C07289=1093.680,277.101,420.370,177.448,19.985,152.800
C07290=1093.686,277.349,420.342,177.452,19.987,152.800
C07291=1093.691,277.598,420.313,177.455,19.990,152.800
C07292=1093.697,277.846,420.284,177.458,19.993,152.800
C07293=1093.703,278.093,420.255,177.461,19.995,152.800
C07294=1093.708,278.342,420.226,177.465,19.997,152.800
C07295=1093.714,278.591,420.197,177.468,20.000,152.800
C07296=1093.719,278.838,420.168,177.470,20.001,152.800
C07297=1093.725,279.087,420.139,177.473,20.004,152.800
C07298=1093.731,279.335,420.110,177.476,20.007,152.800
C07299=1093.737,279.584,420.081,177.480,20.009,152.800
C07300=1093.742,279.831,420.052,177.483,20.011,152.800
C07301=1093.748,280.080,420.023,177.486,20.014,152.800
C07302=1093.754,280.328,419.994,177.489,20.016,152.800
C07303=1093.759,280.576,419.965,177.493,20.018,152.800
C07304=1093.765,280.824,419.936,177.496,20.021,152.800
C07305=1093.770,281.073,419.907,177.499,20.023,152.800
C07306=1093.777,281.321,419.878,177.501,20.025,152.800
C07307=1093.781,281.569,419.849,177.505,20.028,152.800
C07308=1093.788,281.817,419.819,177.508,20.030,152.800
C07309=1093.793,282.066,419.790,177.511,20.032,152.800
C07310=1093.799,282.314,419.760,177.514,20.035,152.800
C07311=1093.804,282.561,419.732,177.517,20.038,152.800
C07312=1093.810,282.810,419.702,177.520,20.040,152.800
C07313=1093.815,283.058,419.672,177.524,20.043,152.800
C07314=1093.821,283.307,419.644,177.527,20.045,152.800
C07315=1093.826,283.555,419.615,177.530,20.047,152.800
C07316=1093.832,283.803,419.585,177.533,20.050,152.800
C07317=1093.838,284.051,419.556,177.536,20.052,152.800
C07318=1093.843,284.285,419.528,177.539,20.055,152.800
C07319=1093.849,284.520,419.501,177.542,20.057,152.800
C07320=1093.854,284.754,419.472,177.545,20.059,152.800
C07321=1093.859,284.988,419.445,177.547,20.061,152.800
C07322=1093.864,285.222,419.417,177.551,20.064,152.800
C07323=1093.870,285.456,419.389,177.554,20.066,152.800
C07324=1093.875,285.691,419.361,177.557,20.068,152.800
C07325=1093.881,285.925,419.333,177.559,20.070,152.800
C07326=1093.886,286.173,419.304,177.563,20.073,152.800
C07327=1093.892,286.421,419.274,177.566,20.076,152.800
C07328=1093.898,286.669,419.245,177.569,20.078,152.800
C07329=1093.903,286.918,419.216,177.572,20.080,152.800
C07330=1093.909,287.166,419.186,177.575,20.083,152.800
C07331=1093.915,287.414,419.156,177.578,20.085,152.800
C07332=1093.921,287.662,419.127,177.582,20.088,152.800
C07333=1093.927,287.911,419.097,177.585,20.091,152.800
C07334=1093.931,288.158,419.068,177.588,20.093,152.800
C07335=1093.937,288.407,419.038,177.591,20.095,152.800
C07336=1093.943,288.654,419.008,177.594,20.098,152.800
C07337=1093.949,288.903,418.979,177.598,20.100,152.800
C07338=1093.958,289.278,418.934,177.602,20.104,152.800
C07339=1093.966,289.653,418.888,177.607,20.108,152.801
C07340=1093.975,290.029,418.843,177.612,20.112,152.801
C07341=1093.983,290.404,418.799,177.616,20.116,152.801
C07342=1093.989,290.652,418.769,177.619,20.118,152.801
C07343=1093.994,290.900,418.739,177.623,20.121,152.801
C07344=1094.001,291.149,418.710,177.626,20.123,152.801
C07345=1094.006,291.396,418.680,177.629,20.126,152.801
C07346=1094.012,291.645,418.650,177.632,20.128,152.801
C07347=1094.018,291.893,418.620,177.635,20.131,152.801
C07348=1094.023,292.141,418.590,177.638,20.134,152.801
C07349=1094.029,292.389,418.560,177.641,20.136,152.801
C07350=1094.035,292.637,418.530,177.645,20.139,152.801
C07351=1094.040,292.885,418.500,177.648,20.141,152.801
C07352=1094.046,293.134,418.470,177.651,20.144,152.801
C07353=1094.052,293.381,418.440,177.654,20.146,152.801
C07354=1094.057,293.630,418.410,177.657,20.149,152.801
C07355=1094.063,293.878,418.380,177.660,20.152,152.801
C07356=1094.069,294.126,418.350,177.663,20.154,152.802
C07357=1094.074,294.374,418.320,177.667,20.157,152.802
C07358=1094.080,294.622,418.290,177.670,20.159,152.802
C07359=1094.086,294.870,418.260,177.673,20.162,152.802
C07360=1094.091,295.118,418.229,177.676,20.164,152.802
C07361=1094.097,295.366,418.200,177.679,20.167,152.802
C07362=1094.103,295.614,418.169,177.682,20.169,152.802
C07363=1094.109,295.862,418.139,177.685,20.172,152.802
C07364=1094.114,296.111,418.109,177.689,20.175,152.802
C07365=1094.119,296.359,418.078,177.692,20.177,152.802
C07366=1094.125,296.606,418.048,177.695,20.180,152.802
C07367=1094.131,296.855,418.018,177.698,20.183,152.802
C07368=1094.136,297.103,417.988,177.701,20.185,152.802
C07369=1094.142,297.351,417.958,177.704,20.188,152.802
C07370=1094.148,297.598,417.927,177.707,20.190,152.802
C07371=1094.154,297.846,417.897,177.710,20.193,152.802
C07372=1094.159,298.095,417.867,177.713,20.196,152.803
C07373=1094.164,298.343,417.836,177.716,20.199,152.803
C07374=1094.170,298.591,417.806,177.720,20.201,152.803
C07375=1094.176,298.838,417.776,177.723,20.204,152.803
C07376=1094.181,299.087,417.745,177.726,20.207,152.803
C07377=1094.188,299.335,417.714,177.729,20.209,152.803
C07378=1094.193,299.584,417.684,177.732,20.212,152.803
C07379=1094.198,299.832,417.653,177.735,20.215,152.803
C07380=1094.204,300.079,417.623,177.738,20.217,152.803
C07381=1094.209,300.328,417.592,177.741,20.220,152.804
C07382=1094.215,300.575,417.562,177.744,20.223,152.804
C07383=1094.221,300.823,417.531,177.748,20.226,152.804
C07384=1094.226,301.071,417.501,177.751,20.229,152.804
C07385=1094.232,301.319,417.470,177.754,20.232,152.804
C07386=1094.237,301.567,417.440,177.757,20.234,152.804
C07387=1094.242,301.815,417.409,177.760,20.237,152.804
C07388=1094.248,302.063,417.379,177.763,20.240,152.804
C07389=1094.253,302.311,417.348,177.766,20.242,152.804
C07390=1094.262,302.700,417.299,177.771,20.247,152.805
C07391=1094.271,303.089,417.251,177.776,20.251,152.805
C07392=1094.280,303.479,417.203,177.781,20.255,152.805
C07393=1094.289,303.869,417.154,177.786,20.260,152.805
C07394=1094.295,304.116,417.124,177.789,20.263,152.805
C07395=1094.300,304.365,417.093,177.792,20.266,152.805
C07396=1094.306,304.612,417.062,177.795,20.269,152.805
C07397=1094.312,304.860,417.031,177.798,20.271,152.806
C07398=1094.318,305.108,417.000,177.802,20.274,152.806
C07399=1094.323,305.357,416.969,177.804,20.277,152.806
C07400=1094.329,305.604,416.939,177.808,20.279,152.806
C07401=1094.334,305.852,416.907,177.811,20.283,152.806
C07402=1094.340,306.100,416.877,177.815,20.285,152.806
C07403=1094.346,306.349,416.846,177.817,20.288,152.806
C07404=1094.352,306.596,416.815,177.821,20.291,152.806
C07405=1094.357,306.844,416.784,177.824,20.294,152.807
C07406=1094.363,307.092,416.753,177.827,20.296,152.807
C07407=1094.369,307.340,416.721,177.830,20.299,152.807
C07408=1094.375,307.588,416.691,177.833,20.302,152.807
C07409=1094.380,307.836,416.660,177.836,20.306,152.807
C07410=1094.386,308.084,416.628,177.840,20.308,152.807
C07411=1094.391,308.332,416.598,177.843,20.311,152.807
C07412=1094.397,308.579,416.566,177.846,20.314,152.807
C07413=1094.403,308.828,416.535,177.849,20.317,152.808
C07414=1094.408,309.076,416.504,177.852,20.319,152.808
C07415=1094.414,309.323,416.473,177.855,20.322,152.808
C07416=1094.420,309.572,416.442,177.858,20.325,152.808
C07417=1094.426,309.820,416.410,177.862,20.328,152.808
C07418=1094.431,310.067,416.380,177.865,20.331,152.808
C07419=1094.437,310.316,416.348,177.868,20.334,152.808
C07420=1094.443,310.563,416.318,177.871,20.336,152.808
C07421=1094.449,310.811,416.286,177.874,20.339,152.809
C07422=1094.454,311.059,416.254,177.877,20.342,152.809
C07423=1094.460,311.307,416.224,177.880,20.345,152.809
C07424=1094.466,311.555,416.192,177.884,20.348,152.809
C07425=1094.471,311.803,416.161,177.887,20.351,152.809
C07426=1094.478,312.051,416.130,177.890,20.354,152.809
C07427=1094.483,312.299,416.097,177.893,20.357,152.809
C07428=1094.489,312.547,416.067,177.896,20.360,152.810
C07429=1094.495,312.795,416.035,177.899,20.363,152.810
C07430=1094.501,313.042,416.003,177.902,20.365,152.810
C07431=1094.506,313.291,415.972,177.906,20.369,152.810
C07432=1094.512,313.538,415.941,177.909,20.371,152.810
C07433=1094.518,313.787,415.909,177.912,20.374,152.810
C07434=1094.524,314.035,415.878,177.915,20.377,152.810
C07435=1094.530,314.283,415.847,177.918,20.380,152.811
C07436=1094.536,314.530,415.815,177.921,20.383,152.811
C07437=1094.542,314.778,415.783,177.924,20.386,152.811
C07438=1094.547,315.026,415.751,177.928,20.389,152.811
C07439=1094.553,315.274,415.721,177.931,20.392,152.811
C07440=1094.559,315.522,415.689,177.933,20.395,152.811
C07441=1094.565,315.770,415.657,177.936,20.398,152.812
C07442=1094.573,316.161,415.607,177.942,20.403,152.812
C07443=1094.582,316.554,415.556,177.947,20.408,152.812
C07444=1094.590,316.945,415.506,177.951,20.413,152.813
C07445=1094.599,317.337,415.456,177.956,20.418,152.813
C07446=1094.605,317.586,415.424,177.959,20.421,152.813
C07447=1094.611,317.833,415.392,177.962,20.424,152.813
C07448=1094.616,318.081,415.360,177.965,20.427,152.813
C07449=1094.622,318.329,415.328,177.969,20.430,152.814
C07450=1094.627,318.576,415.297,177.972,20.433,152.814
C07451=1094.633,318.825,415.265,177.975,20.436,152.814
C07452=1094.639,319.072,415.233,177.978,20.439,152.814
C07453=1094.644,319.321,415.200,177.981,20.442,152.815
C07454=1094.650,319.569,415.168,177.984,20.446,152.815
C07455=1094.655,319.816,415.137,177.987,20.449,152.815
C07456=1094.661,320.065,415.105,177.990,20.452,152.815
C07457=1094.667,320.312,415.073,177.993,20.455,152.815
C07458=1094.673,320.560,415.041,177.997,20.459,152.816
C07459=1094.678,320.808,415.009,178.000,20.462,152.816
C07460=1094.683,321.056,414.977,178.002,20.465,152.816
C07461=1094.689,321.303,414.944,178.005,20.468,152.816
C07462=1094.695,321.551,414.912,178.009,20.471,152.816
C07463=1094.701,321.800,414.880,178.012,20.474,152.817
C07464=1094.707,322.047,414.849,178.015,20.477,152.817
C07465=1094.712,322.295,414.817,178.018,20.481,152.817
C07466=1094.717,322.543,414.784,178.022,20.484,152.817
C07467=1094.723,322.791,414.752,178.024,20.487,152.818
C07468=1094.729,323.039,414.720,178.027,20.490,152.818
C07469=1094.735,323.287,414.688,178.030,20.493,152.818
C07470=1094.741,323.534,414.655,178.034,20.497,152.818
C07471=1094.746,323.783,414.623,178.037,20.500,152.819
C07472=1094.752,324.030,414.591,178.040,20.503,152.819
C07473=1094.758,324.278,414.558,178.043,20.506,152.819
C07474=1094.764,324.526,414.526,178.046,20.510,152.819
C07475=1094.769,324.774,414.494,178.049,20.513,152.820
C07476=1094.775,325.021,414.461,178.052,20.516,152.820
C07477=1094.781,325.270,414.429,178.055,20.519,152.820
C07478=1094.787,325.517,414.396,178.059,20.523,152.820
C07479=1094.792,325.765,414.364,178.062,20.526,152.820
C07480=1094.798,326.013,414.332,178.064,20.529,152.821
C07481=1094.804,326.261,414.299,178.068,20.533,152.821
C07482=1094.809,326.509,414.267,178.071,20.536,152.821
C07483=1094.815,326.756,414.234,178.074,20.539,152.821
C07484=1094.821,327.004,414.202,178.077,20.542,152.822
C07485=1094.827,327.252,414.169,178.080,20.546,152.822
C07486=1094.833,327.501,414.137,178.083,20.549,152.822
C07487=1094.838,327.747,414.105,178.086,20.552,152.822
C07488=1094.844,327.995,414.071,178.090,20.556,152.823
C07489=1094.850,328.244,414.039,178.093,20.559,152.823
C07490=1094.856,328.491,414.006,178.096,20.562,152.823
C07491=1094.861,328.740,413.974,178.099,20.566,152.823
C07492=1094.867,328.987,413.942,178.102,20.569,152.824
C07493=1094.873,329.234,413.909,178.105,20.572,152.824
C07494=1094.882,329.619,413.858,178.110,20.577,152.824
C07495=1094.891,330.004,413.807,178.115,20.583,152.825
C07496=1094.900,330.389,413.757,178.119,20.588,152.825
C07497=1094.909,330.774,413.705,178.124,20.593,152.826
C07498=1094.915,331.022,413.673,178.127,20.596,152.826
C07499=1094.921,331.269,413.640,178.131,20.600,152.826
C07500=1094.927,331.518,413.607,178.134,20.603,152.826
C07501=1094.933,331.766,413.575,178.137,20.607,152.827
C07502=1094.939,332.014,413.541,178.140,20.610,152.827
C07503=1094.945,332.261,413.508,178.143,20.614,152.827
C07504=1094.950,332.509,413.475,178.146,20.617,152.828
C07505=1094.956,332.757,413.443,178.150,20.621,152.828
C07506=1094.961,333.004,413.410,178.152,20.624,152.828
C07507=1094.967,333.252,413.377,178.156,20.628,152.829
C07508=1094.973,333.500,413.344,178.159,20.631,152.829
C07509=1094.979,333.748,413.311,178.162,20.634,152.829
C07510=1094.984,333.996,413.277,178.165,20.638,152.829
C07511=1094.991,334.243,413.245,178.168,20.642,152.830
C07512=1094.996,334.491,413.211,178.171,20.645,152.830
C07513=1095.002,334.739,413.178,178.174,20.649,152.830
C07514=1095.007,334.986,413.145,178.177,20.652,152.831
C07515=1095.013,335.234,413.112,178.181,20.656,152.831
C07516=1095.019,335.482,413.079,178.183,20.660,152.831
C07517=1095.024,335.730,413.046,178.186,20.663,152.832
C07518=1095.030,335.977,413.013,178.190,20.667,152.832
C07519=1095.036,336.225,412.980,178.192,20.670,152.832
C07520=1095.041,336.473,412.946,178.196,20.674,152.833
C07521=1095.047,336.721,412.913,178.199,20.677,152.833
C07522=1095.053,336.969,412.880,178.202,20.681,152.833
C07523=1095.059,337.216,412.846,178.205,20.685,152.834
C07524=1095.065,337.464,412.813,178.208,20.688,152.834
C07525=1095.070,337.712,412.779,178.212,20.692,152.834
C07526=1095.077,337.959,412.747,178.214,20.695,152.835
C07527=1095.082,338.207,412.713,178.217,20.699,152.835
C07528=1095.088,338.455,412.680,178.221,20.703,152.835
C07529=1095.094,338.702,412.646,178.223,20.706,152.836
C07530=1095.099,338.950,412.613,178.227,20.710,152.836
C07531=1095.105,339.198,412.579,178.230,20.714,152.836
C07532=1095.110,339.446,412.546,178.233,20.718,152.837
C07533=1095.116,339.693,412.512,178.236,20.721,152.837
C07534=1095.122,339.941,412.479,178.239,20.725,152.838
C07535=1095.128,340.189,412.446,178.242,20.729,152.838
C07536=1095.134,340.436,412.412,178.245,20.732,152.838
C07537=1095.139,340.684,412.378,178.248,20.736,152.839
C07538=1095.145,340.932,412.345,178.251,20.740,152.839
C07539=1095.151,341.179,412.311,178.254,20.744,152.840
C07540=1095.156,341.427,412.278,178.257,20.747,152.840
C07541=1095.162,341.674,412.244,178.261,20.751,152.840
C07542=1095.168,341.922,412.210,178.263,20.755,152.841
C07543=1095.174,342.170,412.176,178.267,20.759,152.841
C07544=1095.180,342.418,412.142,178.269,20.763,152.841
C07545=1095.186,342.666,412.108,178.273,20.767,152.842
C07546=1095.194,343.045,412.057,178.278,20.773,152.843
C07547=1095.203,343.424,412.005,178.282,20.778,152.843
C07548=1095.212,343.803,411.954,178.287,20.784,152.844
C07549=1095.220,344.181,411.902,178.291,20.790,152.844
C07550=1095.226,344.429,411.868,178.295,20.794,152.845
C07551=1095.232,344.677,411.834,178.297,20.798,152.845
C07552=1095.238,344.924,411.800,178.301,20.802,152.845
C07553=1095.244,345.172,411.766,178.304,20.806,152.846
C07554=1095.249,345.420,411.733,178.307,20.810,152.846
C07555=1095.255,345.667,411.699,178.310,20.813,152.847
C07556=1095.261,345.914,411.665,178.313,20.817,152.847
C07557=1095.267,346.163,411.630,178.316,20.821,152.848
C07558=1095.272,346.410,411.596,178.319,20.826,152.848
C07559=1095.278,346.658,411.562,178.322,20.829,152.849
C07560=1095.284,346.905,411.528,178.325,20.833,152.849
C07561=1095.290,347.152,411.494,178.328,20.837,152.849
C07562=1095.295,347.401,411.460,178.331,20.841,152.850
C07563=1095.301,347.649,411.426,178.335,20.846,152.850
C07564=1095.307,347.896,411.392,178.337,20.849,152.851
C07565=1095.313,348.143,411.358,178.341,20.853,152.851
C07566=1095.318,348.391,411.323,178.343,20.857,152.852
C07567=1095.324,348.638,411.289,178.347,20.862,152.852
C07568=1095.330,348.887,411.255,178.349,20.865,152.852
C07569=1095.335,349.134,411.221,178.353,20.869,152.853
C07570=1095.341,349.381,411.187,178.355,20.873,152.853
C07571=1095.347,349.629,411.153,178.359,20.878,152.854
C07572=1095.352,349.877,411.118,178.362,20.882,152.854
C07573=1095.358,350.124,411.084,178.365,20.886,152.855
C07574=1095.364,350.372,411.050,178.368,20.890,152.855
C07575=1095.369,350.619,411.015,178.371,20.894,152.856
C07576=1095.376,350.867,410.981,178.374,20.898,152.856
C07577=1095.382,351.114,410.946,178.378,20.902,152.857
C07578=1095.387,351.362,410.912,178.380,20.906,152.857
C07579=1095.393,351.609,410.878,178.383,20.911,152.858
C07580=1095.399,351.857,410.843,178.386,20.915,152.858
C07581=1095.404,352.104,410.808,178.389,20.919,152.859
C07582=1095.410,352.352,410.774,178.393,20.923,152.859
C07583=1095.416,352.600,410.739,178.395,20.927,152.860
C07584=1095.422,352.847,410.705,178.399,20.931,152.860
C07585=1095.428,353.094,410.671,178.401,20.935,152.861
C07586=1095.433,353.343,410.636,178.405,20.940,152.861
C07587=1095.440,353.589,410.601,178.408,20.944,152.862
C07588=1095.445,353.837,410.566,178.410,20.948,152.862
C07589=1095.451,354.085,410.532,178.414,20.953,152.863
C07590=1095.456,354.333,410.497,178.416,20.957,152.863
C07591=1095.463,354.579,410.463,178.420,20.961,152.864
C07592=1095.468,354.828,410.428,178.423,20.966,152.864
C07593=1095.473,355.075,410.393,178.425,20.970,152.865
C07594=1095.480,355.322,410.358,178.429,20.974,152.865
C07595=1095.485,355.570,410.323,178.432,20.978,152.866
C07596=1095.491,355.817,410.289,178.434,20.983,152.867
C07597=1095.497,356.064,410.254,178.438,20.987,152.867
C07598=1095.505,356.447,410.200,178.442,20.994,152.868
C07599=1095.514,356.828,410.146,178.447,21.000,152.869
C07600=1095.524,357.209,410.093,178.452,21.008,152.870
C07601=1095.532,357.590,410.039,178.457,21.014,152.870
C07602=1095.538,357.838,410.003,178.459,21.018,152.871
C07603=1095.544,358.085,409.969,178.462,21.023,152.872
C07604=1095.550,358.333,409.934,178.465,21.027,152.872
C07605=1095.555,358.580,409.899,178.468,21.031,152.873
C07606=1095.561,358.827,409.864,178.471,21.036,152.873
C07607=1095.567,359.075,409.829,178.475,21.040,152.874
C07608=1095.573,359.322,409.794,178.478,21.045,152.874
C07609=1095.579,359.570,409.759,178.480,21.050,152.875
C07610=1095.584,359.817,409.724,178.483,21.054,152.876
C07611=1095.590,360.065,409.688,178.487,21.059,152.876
C07612=1095.596,360.312,409.653,178.489,21.063,152.877
C07613=1095.602,360.560,409.619,178.492,21.067,152.877
C07614=1095.608,360.807,409.583,178.496,21.072,152.878
C07615=1095.614,361.055,409.547,178.499,21.077,152.879
C07616=1095.619,361.302,409.513,178.501,21.081,152.879
C07617=1095.625,361.550,409.477,178.504,21.086,152.880
C07618=1095.630,361.797,409.442,178.507,21.091,152.880
C07619=1095.637,362.044,409.407,178.510,21.095,152.881
C07620=1095.643,362.291,409.371,178.513,21.099,152.882
C07621=1095.648,362.539,409.336,178.516,21.104,152.882
C07622=1095.654,362.786,409.301,178.520,21.109,152.883
C07623=1095.660,363.034,409.265,178.522,21.113,152.883
C07624=1095.665,363.281,409.230,178.525,21.118,152.884
C07625=1095.672,363.528,409.195,178.528,21.123,152.885
C07626=1095.677,363.775,409.159,178.532,21.128,152.885
C07627=1095.683,364.023,409.124,178.534,21.132,152.886
C07628=1095.689,364.271,409.088,178.537,21.137,152.887
C07629=1095.695,364.518,409.052,178.540,21.142,152.887
C07630=1095.701,364.765,409.017,178.543,21.146,152.888
C07631=1095.706,365.012,408.981,178.546,21.152,152.889
C07632=1095.712,365.260,408.946,178.549,21.156,152.889
C07633=1095.718,365.507,408.910,178.552,21.161,152.890
C07634=1095.724,365.755,408.875,178.555,21.165,152.891
C07635=1095.730,366.002,408.839,178.558,21.170,152.891
C07636=1095.735,366.249,408.803,178.560,21.175,152.892
C07637=1095.741,366.497,408.768,178.564,21.180,152.893
C07638=1095.747,366.744,408.732,178.567,21.185,152.893
C07639=1095.753,366.992,408.697,178.570,21.190,152.894
C07640=1095.758,367.239,408.661,178.573,21.195,152.895
C07641=1095.764,367.486,408.626,178.575,21.199,152.895
C07642=1095.770,367.734,408.588,178.578,21.204,152.896
C07643=1095.775,367.981,408.553,178.581,21.209,152.897
C07644=1095.781,368.228,408.517,178.585,21.214,152.897
C07645=1095.787,368.476,408.482,178.588,21.219,152.898
C07646=1095.793,368.723,408.446,178.591,21.224,152.899
C07647=1095.799,368.970,408.410,178.593,21.229,152.900
C07648=1095.805,369.217,408.374,178.596,21.234,152.900
C07649=1095.810,369.465,408.338,178.599,21.239,152.901
C07650=1095.820,369.861,408.280,178.604,21.247,152.902
C07651=1095.829,370.258,408.223,178.609,21.255,152.903
C07652=1095.838,370.655,408.165,178.613,21.263,152.905
C07653=1095.848,371.051,408.107,178.618,21.271,152.906
C07654=1095.854,371.298,408.071,178.621,21.276,152.907
C07655=1095.859,371.545,408.035,178.624,21.281,152.907
C07656=1095.865,371.793,407.999,178.627,21.287,152.908
C07657=1095.871,372.040,407.963,178.630,21.291,152.909
C07658=1095.877,372.287,407.927,178.633,21.297,152.910
C07659=1095.882,372.534,407.890,178.635,21.301,152.910
C07660=1095.888,372.782,407.854,178.638,21.307,152.911
C07661=1095.895,373.029,407.818,178.641,21.312,152.912
C07662=1095.901,373.276,407.782,178.644,21.317,152.913
C07663=1095.906,373.524,407.745,178.647,21.322,152.913
C07664=1095.912,373.771,407.710,178.650,21.327,152.914
C07665=1095.918,374.018,407.673,178.653,21.333,152.915
C07666=1095.924,374.265,407.636,178.656,21.338,152.916
C07667=1095.930,374.513,407.601,178.659,21.343,152.916
C07668=1095.935,374.759,407.565,178.662,21.349,152.917
C07669=1095.941,375.006,407.528,178.665,21.354,152.918
C07670=1095.947,375.254,407.491,178.667,21.359,152.919
C07671=1095.953,375.502,407.455,178.670,21.364,152.920
C07672=1095.958,375.748,407.419,178.673,21.369,152.921
C07673=1095.964,375.995,407.382,178.676,21.375,152.922
C07674=1095.970,376.242,407.345,178.679,21.380,152.922
C07675=1095.976,376.490,407.309,178.682,21.386,152.923
C07676=1095.982,376.737,407.272,178.685,21.391,152.924
C07677=1095.987,376.984,407.236,178.688,21.397,152.925
C07678=1095.993,377.231,407.199,178.691,21.402,152.926
C07679=1095.999,377.478,407.162,178.693,21.408,152.927
C07680=1096.005,377.725,407.126,178.696,21.413,152.927
C07681=1096.011,377.973,407.089,178.699,21.418,152.928
C07682=1096.017,378.220,407.052,178.702,21.424,152.929
C07683=1096.022,378.467,407.016,178.705,21.429,152.930
C07684=1096.027,378.715,406.979,178.708,21.435,152.931
C07685=1096.034,378.962,406.943,178.711,21.441,152.932
C07686=1096.039,379.209,406.906,178.714,21.446,152.933
C07687=1096.046,379.456,406.869,178.717,21.451,152.933
C07688=1096.051,379.703,406.832,178.719,21.457,152.934
C07689=1096.058,379.950,406.795,178.722,21.463,152.935
C07690=1096.063,380.197,406.758,178.725,21.468,152.936
C07691=1096.069,380.445,406.721,178.728,21.473,152.937
C07692=1096.075,380.692,406.685,178.731,21.479,152.938
C07693=1096.081,380.939,406.648,178.734,21.485,152.939
C07694=1096.087,381.185,406.612,178.737,21.490,152.940
C07695=1096.092,381.433,406.575,178.739,21.496,152.941
C07696=1096.098,381.680,406.537,178.742,21.502,152.942
C07697=1096.105,381.926,406.500,178.745,21.507,152.942
C07698=1096.110,382.174,406.463,178.748,21.513,152.943
C07699=1096.116,382.421,406.426,178.751,21.518,152.944
C07700=1096.122,382.668,406.390,178.753,21.525,152.945
C07701=1096.128,382.915,406.352,178.756,21.530,152.946
C07702=1096.133,383.127,406.320,178.759,21.535,152.947
C07703=1096.138,383.339,406.289,178.761,21.540,152.948
C07704=1096.143,383.551,406.256,178.763,21.545,152.949
C07705=1096.148,383.763,406.225,178.766,21.550,152.950
C07706=1096.153,383.975,406.192,178.768,21.555,152.950
C07707=1096.158,384.187,406.161,178.771,21.560,152.951
C07708=1096.163,384.399,406.129,178.774,21.565,152.952
C07709=1096.168,384.610,406.097,178.776,21.570,152.953
C07710=1096.173,384.858,406.060,178.779,21.576,152.954
C07711=1096.179,385.104,406.022,178.781,21.582,152.955
C07712=1096.185,385.352,405.985,178.784,21.588,152.956
C07713=1096.191,385.599,405.948,178.788,21.594,152.957
C07714=1096.197,385.846,405.911,178.790,21.600,152.958
C07715=1096.202,386.093,405.874,178.793,21.606,152.959
C07716=1096.208,386.340,405.836,178.796,21.612,152.960
C07717=1096.214,386.587,405.799,178.798,21.618,152.961
C07718=1096.220,386.834,405.761,178.801,21.624,152.962
C07719=1096.226,387.081,405.723,178.804,21.630,152.963
C07720=1096.232,387.329,405.686,178.807,21.637,152.964
C07721=1096.238,387.575,405.648,178.810,21.643,152.965
C07722=1096.244,387.822,405.610,178.813,21.648,152.966
C07723=1096.249,388.070,405.573,178.815,21.654,152.967
C07724=1096.255,388.316,405.536,178.818,21.660,152.968
C07725=1096.261,388.563,405.498,178.821,21.666,152.969
C07726=1096.267,388.810,405.461,178.824,21.673,152.970
C07727=1096.273,389.057,405.423,178.827,21.679,152.971
C07728=1096.279,389.304,405.385,178.829,21.685,152.972
C07729=1096.285,389.551,405.347,178.832,21.691,152.973
C07730=1096.291,389.799,405.310,178.835,21.698,152.975
C07731=1096.297,390.045,405.272,178.838,21.704,152.976
C07732=1096.303,390.292,405.235,178.841,21.710,152.977
C07733=1096.308,390.539,405.197,178.843,21.717,152.978
C07734=1096.314,390.786,405.159,178.846,21.723,152.979
C07735=1096.321,391.033,405.121,178.849,21.729,152.980
C07736=1096.326,391.280,405.084,178.852,21.736,152.981
C07737=1096.332,391.527,405.046,178.855,21.742,152.982
C07738=1096.338,391.774,405.008,178.857,21.748,152.983
C07739=1096.345,392.021,404.970,178.860,21.754,152.984
C07740=1096.351,392.268,404.933,178.862,21.760,152.985
C07741=1096.357,392.515,404.895,178.866,21.767,152.987
C07742=1096.362,392.762,404.856,178.868,21.774,152.988
C07743=1096.368,393.009,404.819,178.871,21.780,152.989
C07744=1096.374,393.256,404.781,178.873,21.786,152.990
C07745=1096.380,393.503,404.743,178.877,21.793,152.991
C07746=1096.385,393.750,404.704,178.879,21.800,152.992
C07747=1096.392,393.997,404.666,178.882,21.806,152.994
C07748=1096.398,394.244,404.629,178.884,21.812,152.995
C07749=1096.403,394.491,404.590,178.888,21.819,152.996
C07750=1096.409,394.737,404.552,178.890,21.826,152.997
C07751=1096.415,394.985,404.514,178.892,21.832,152.998
C07752=1096.421,395.231,404.476,178.896,21.839,153.000
C07753=1096.427,395.479,404.438,178.898,21.846,153.001
C07754=1096.433,395.726,404.399,178.901,21.852,153.002
C07755=1096.439,395.972,404.360,178.903,21.859,153.003
C07756=1096.444,396.219,404.323,178.906,21.866,153.004
C07757=1096.451,396.467,404.284,178.909,21.872,153.006
C07758=1096.456,396.685,404.250,178.912,21.878,153.007
C07759=1096.461,396.903,404.217,178.914,21.885,153.008
C07760=1096.466,397.121,404.183,178.916,21.890,153.009
C07761=1096.472,397.339,404.149,178.919,21.896,153.010
C07762=1096.476,397.557,404.114,178.921,21.903,153.011
C07763=1096.482,397.776,404.080,178.923,21.908,153.012
C07764=1096.487,397.994,404.047,178.926,21.915,153.013
C07765=1096.492,398.213,404.013,178.928,21.921,153.014
C07766=1096.498,398.460,403.974,178.931,21.928,153.016
C07767=1096.504,398.707,403.936,178.934,21.935,153.017
C07768=1096.510,398.953,403.897,178.936,21.942,153.018
C07769=1096.516,399.200,403.859,178.939,21.948,153.020
C07770=1096.522,399.447,403.820,178.942,21.956,153.021
C07771=1096.528,399.695,403.781,178.944,21.962,153.022
C07772=1096.534,399.941,403.743,178.948,21.970,153.023
C07773=1096.540,400.189,403.704,178.950,21.976,153.025
C07774=1096.546,400.435,403.666,178.952,21.983,153.026
C07775=1096.551,400.682,403.627,178.955,21.991,153.027
C07776=1096.557,400.929,403.588,178.957,21.998,153.029
C07777=1096.564,401.176,403.549,178.961,22.005,153.030
C07778=1096.569,401.423,403.511,178.963,22.012,153.031
C07779=1096.575,401.670,403.471,178.966,22.020,153.033
C07780=1096.581,401.916,403.433,178.968,22.027,153.034
C07781=1096.587,402.164,403.394,178.971,22.034,153.036
C07782=1096.592,402.410,403.355,178.974,22.041,153.037
C07783=1096.599,402.657,403.316,178.976,22.048,153.038
C07784=1096.604,402.904,403.278,178.979,22.056,153.040
C07785=1096.611,403.151,403.238,178.981,22.063,153.041
C07786=1096.616,403.398,403.199,178.985,22.070,153.042
C07787=1096.623,403.644,403.160,178.987,22.078,153.044
C07788=1096.628,403.891,403.121,178.990,22.085,153.045
C07789=1096.634,404.139,403.083,178.992,22.092,153.047
C07790=1096.641,404.385,403.044,178.995,22.100,153.048
C07791=1096.646,404.632,403.005,178.997,22.107,153.050
C07792=1096.652,404.879,402.965,179.001,22.115,153.051
C07793=1096.658,405.125,402.926,179.003,22.122,153.052
C07794=1096.664,405.373,402.887,179.006,22.130,153.054
C07795=1096.670,405.620,402.847,179.009,22.138,153.055
C07796=1096.676,405.866,402.809,179.011,22.145,153.057
C07797=1096.682,406.113,402.769,179.014,22.153,153.058
C07798=1096.688,406.360,402.730,179.016,22.160,153.060
C07799=1096.694,406.607,402.691,179.019,22.168,153.061
C07800=1096.700,406.854,402.652,179.022,22.176,153.063
C07801=1096.705,407.100,402.612,179.024,22.183,153.064
C07802=1096.711,407.347,402.573,179.027,22.191,153.066
C07803=1096.718,407.594,402.534,179.029,22.199,153.067
C07804=1096.724,407.842,402.494,179.032,22.207,153.069
C07805=1096.729,408.087,402.454,179.035,22.215,153.070
C07806=1096.735,408.334,402.415,179.037,22.222,153.072
C07807=1096.742,408.582,402.376,179.040,22.231,153.073
C07808=1096.747,408.828,402.336,179.043,22.238,153.075
C07809=1096.753,409.075,402.297,179.045,22.246,153.076
C07810=1096.759,409.322,402.257,179.048,22.254,153.078
C07811=1096.765,409.568,402.218,179.051,22.263,153.080
C07812=1096.770,409.816,402.178,179.053,22.270,153.081
C07813=1096.777,410.062,402.138,179.056,22.278,153.083
C07814=1096.781,410.281,402.103,179.058,22.285,153.084
C07815=1096.787,410.499,402.068,179.060,22.292,153.086
C07816=1096.792,410.718,402.033,179.063,22.300,153.087
C07817=1096.797,410.936,401.998,179.065,22.307,153.088
C07818=1096.803,411.155,401.962,179.067,22.314,153.090
C07819=1096.808,411.373,401.928,179.070,22.322,153.091
C07820=1096.813,411.592,401.892,179.072,22.329,153.093
C07821=1096.818,411.810,401.857,179.075,22.336,153.094
C07822=1096.825,412.057,401.817,179.077,22.344,153.096
C07823=1096.831,412.304,401.777,179.079,22.352,153.097
C07824=1096.837,412.551,401.738,179.082,22.361,153.099
C07825=1096.843,412.798,401.697,179.085,22.369,153.101
C07826=1096.848,413.043,401.657,179.088,22.377,153.102
C07827=1096.854,413.290,401.618,179.090,22.385,153.104
C07828=1096.861,413.537,401.578,179.092,22.394,153.106
C07829=1096.867,413.784,401.538,179.095,22.402,153.107
C07830=1096.873,414.031,401.498,179.098,22.411,153.109
C07831=1096.879,414.277,401.457,179.101,22.419,153.111
C07832=1096.885,414.525,401.418,179.104,22.428,153.113
C07833=1096.891,414.771,401.378,179.105,22.436,153.114
C07834=1096.896,415.017,401.337,179.108,22.445,153.116
C07835=1096.903,415.264,401.297,179.111,22.453,153.118
C07836=1096.909,415.511,401.258,179.114,22.462,153.119
C07837=1096.915,415.757,401.218,179.116,22.471,153.121
C07838=1096.921,416.004,401.177,179.119,22.479,153.123
C07839=1096.927,416.251,401.137,179.122,22.488,153.125
C07840=1096.934,416.497,401.097,179.124,22.497,153.126
C07841=1096.939,416.744,401.056,179.127,22.505,153.128
C07842=1096.946,416.991,401.016,179.130,22.514,153.130
C07843=1096.951,417.237,400.975,179.132,22.522,153.132
C07844=1096.957,417.485,400.936,179.134,22.531,153.134
C07845=1096.963,417.731,400.895,179.137,22.541,153.135
C07846=1096.969,417.978,400.855,179.139,22.550,153.137
C07847=1096.975,418.224,400.813,179.142,22.559,153.139
C07848=1096.982,418.471,400.773,179.145,22.568,153.141
C07849=1096.987,418.717,400.733,179.147,22.577,153.143
C07850=1096.993,418.963,400.693,179.150,22.586,153.145
C07851=1096.999,419.210,400.652,179.152,22.595,153.147
C07852=1097.004,419.457,400.611,179.155,22.604,153.148
C07853=1097.011,419.703,400.571,179.158,22.613,153.150
C07854=1097.016,419.950,400.530,179.160,22.622,153.152
C07855=1097.023,420.197,400.490,179.163,22.631,153.154
C07856=1097.029,420.444,400.448,179.166,22.640,153.156
C07857=1097.036,420.690,400.408,179.168,22.650,153.158
C07858=1097.041,420.937,400.367,179.171,22.659,153.160
C07859=1097.047,421.183,400.326,179.174,22.668,153.162
C07860=1097.054,421.430,400.286,179.176,22.677,153.164
C07861=1097.059,421.677,400.245,179.179,22.687,153.166
C07862=1097.066,421.922,400.204,179.181,22.696,153.168
C07863=1097.072,422.169,400.163,179.183,22.706,153.170
C07864=1097.077,422.416,400.123,179.186,22.715,153.172
C07865=1097.084,422.662,400.082,179.188,22.724,153.174
C07866=1097.090,422.909,400.041,179.191,22.734,153.175
C07867=1097.096,423.155,400.000,179.194,22.744,153.177
C07868=1097.101,423.402,399.959,179.197,22.753,153.179
C07869=1097.109,423.648,399.918,179.199,22.763,153.182
C07870=1097.113,423.874,399.880,179.202,22.772,153.183
C07871=1097.119,424.099,399.843,179.203,22.780,153.185
C07872=1097.124,424.325,399.805,179.206,22.789,153.187
C07873=1097.130,424.550,399.768,179.209,22.798,153.189
C07874=1097.136,424.776,399.730,179.210,22.807,153.191
C07875=1097.140,425.002,399.692,179.213,22.816,153.193
C07876=1097.146,425.227,399.655,179.215,22.826,153.195
C07877=1097.152,425.453,399.617,179.217,22.834,153.197
C07878=1097.158,425.700,399.575,179.220,22.845,153.199
C07879=1097.164,425.946,399.534,179.223,22.854,153.201
C07880=1097.170,426.192,399.493,179.225,22.864,153.203
C07881=1097.176,426.439,399.452,179.227,22.874,153.205
C07882=1097.183,426.685,399.410,179.231,22.884,153.207
C07883=1097.189,426.932,399.369,179.233,22.895,153.209
C07884=1097.195,427.178,399.327,179.235,22.904,153.212
C07885=1097.200,427.424,399.286,179.237,22.914,153.214
C07886=1097.207,427.671,399.244,179.240,22.925,153.216
C07887=1097.213,427.917,399.203,179.243,22.935,153.218
C07888=1097.219,428.163,399.161,179.245,22.945,153.220
C07889=1097.225,428.410,399.120,179.248,22.955,153.222
C07890=1097.231,428.657,399.079,179.250,22.966,153.225
C07891=1097.238,428.903,399.038,179.253,22.976,153.227
C07892=1097.243,429.150,398.996,179.256,22.986,153.229
C07893=1097.250,429.396,398.953,179.258,22.997,153.231
C07894=1097.256,429.642,398.912,179.260,23.007,153.234
C07895=1097.262,429.888,398.870,179.263,23.018,153.236
C07896=1097.268,430.134,398.829,179.265,23.028,153.238
C07897=1097.274,430.381,398.787,179.267,23.039,153.240
C07898=1097.280,430.628,398.746,179.270,23.050,153.243
C07899=1097.286,430.874,398.704,179.272,23.060,153.245
C07900=1097.292,431.120,398.661,179.275,23.071,153.247
C07901=1097.298,431.367,398.619,179.277,23.081,153.250
C07902=1097.304,431.613,398.578,179.280,23.092,153.252
C07903=1097.311,431.859,398.535,179.282,23.103,153.254
C07904=1097.317,432.105,398.494,179.284,23.114,153.257
C07905=1097.323,432.351,398.453,179.287,23.125,153.259
C07906=1097.329,432.598,398.409,179.289,23.135,153.262
C07907=1097.335,432.844,398.368,179.292,23.147,153.264
C07908=1097.342,433.091,398.326,179.295,23.157,153.266
C07909=1097.348,433.337,398.284,179.297,23.169,153.269
C07910=1097.353,433.583,398.242,179.299,23.179,153.271
C07911=1097.360,433.830,398.199,179.302,23.191,153.274
C07912=1097.366,434.076,398.158,179.304,23.202,153.276
C07913=1097.372,434.322,398.115,179.307,23.214,153.279
C07914=1097.378,434.569,398.073,179.309,23.224,153.281
C07915=1097.383,434.814,398.031,179.312,23.236,153.284
C07916=1097.390,435.061,397.988,179.314,23.247,153.286
C07917=1097.396,435.307,397.947,179.316,23.259,153.289
C07918=1097.402,435.554,397.903,179.319,23.270,153.291
C07919=1097.409,435.799,397.861,179.321,23.281,153.294
C07920=1097.414,436.046,397.819,179.324,23.293,153.296
C07921=1097.421,436.292,397.777,179.326,23.304,153.299
C07922=1097.426,436.538,397.734,179.328,23.316,153.301
C07923=1097.433,436.784,397.691,179.331,23.328,153.304
C07924=1097.438,437.031,397.649,179.333,23.339,153.307
C07925=1097.445,437.277,397.607,179.336,23.351,153.309
C07926=1097.452,437.568,397.556,179.339,23.365,153.312
C07927=1097.460,437.860,397.506,179.342,23.379,153.315
C07928=1097.467,438.152,397.456,179.344,23.393,153.319
C07929=1097.474,438.443,397.404,179.347,23.407,153.322
C07930=1097.481,438.690,397.362,179.349,23.419,153.324
C07931=1097.487,438.935,397.319,179.352,23.431,153.327
C07932=1097.494,439.182,397.276,179.354,23.443,153.330
C07933=1097.499,439.428,397.234,179.356,23.455,153.332
C07934=1097.505,439.674,397.191,179.359,23.467,153.335
C07935=1097.512,439.920,397.148,179.361,23.479,153.338
C07936=1097.518,440.166,397.105,179.363,23.491,153.341
C07937=1097.525,440.413,397.063,179.366,23.503,153.343
C07938=1097.531,440.659,397.019,179.368,23.516,153.346
C07939=1097.536,440.904,396.976,179.371,23.528,153.349
C07940=1097.543,441.151,396.934,179.372,23.540,153.352
C07941=1097.549,441.397,396.891,179.375,23.553,153.355
C07942=1097.555,441.643,396.847,179.378,23.565,153.357
C07943=1097.561,441.889,396.804,179.380,23.578,153.360
C07944=1097.568,442.135,396.762,179.383,23.591,153.363
C07945=1097.574,442.381,396.718,179.384,23.603,153.366
C07946=1097.580,442.627,396.675,179.387,23.616,153.369
C07947=1097.586,442.873,396.632,179.389,23.628,153.372
C07948=1097.592,443.119,396.588,179.391,23.642,153.375
C07949=1097.599,443.366,396.545,179.394,23.654,153.378
C07950=1097.605,443.611,396.502,179.396,23.667,153.381
C07951=1097.611,443.857,396.459,179.398,23.680,153.384
C07952=1097.617,444.103,396.415,179.400,23.693,153.387
C07953=1097.624,444.349,396.371,179.402,23.706,153.390
C07954=1097.629,444.595,396.328,179.404,23.719,153.393
C07955=1097.636,444.841,396.285,179.405,23.732,153.396
C07956=1097.642,445.088,396.241,179.407,23.744,153.399
C07957=1097.648,445.334,396.198,179.408,23.757,153.402
C07958=1097.655,445.579,396.154,179.410,23.770,153.405
C07959=1097.662,445.826,396.111,179.410,23.783,153.408
C07960=1097.667,446.071,396.068,179.411,23.795,153.411
C07961=1097.673,446.318,396.023,179.412,23.809,153.414
C07962=1097.679,446.564,395.979,179.412,23.821,153.417
C07963=1097.686,446.810,395.936,179.413,23.834,153.421
C07964=1097.692,447.056,395.892,179.413,23.847,153.424
C07965=1097.698,447.302,395.849,179.413,23.859,153.427
C07966=1097.704,447.547,395.805,179.413,23.872,153.430
C07967=1097.711,447.793,395.761,179.413,23.885,153.433
C07968=1097.717,448.039,395.717,179.412,23.897,153.437
C07969=1097.723,448.286,395.674,179.412,23.910,153.440
C07970=1097.730,448.532,395.630,179.412,23.923,153.443
C07971=1097.736,448.778,395.587,179.411,23.936,153.447
C07972=1097.742,449.024,395.542,179.410,23.948,153.450
C07973=1097.748,449.270,395.498,179.409,23.960,153.453
C07974=1097.754,449.515,395.455,179.409,23.973,153.456
C07975=1097.760,449.761,395.411,179.407,23.986,153.460
C07976=1097.767,450.007,395.367,179.406,23.998,153.463
C07977=1097.775,450.254,395.323,179.406,24.010,153.466
C07978=1097.381,450.244,395.165,179.346,24.226,153.529
C07979=1097.374,449.998,395.209,179.346,24.213,153.526
C07980=1097.367,449.752,395.253,179.348,24.201,153.522
C07981=1097.360,449.507,395.297,179.349,24.189,153.519
C07982=1097.354,449.261,395.341,179.350,24.175,153.516
C07983=1097.348,449.015,395.385,179.350,24.163,153.512
C07984=1097.341,448.769,395.429,179.351,24.151,153.509
C07985=1097.335,448.523,395.473,179.352,24.138,153.506
C07986=1097.329,448.277,395.517,179.352,24.125,153.502
C07987=1097.323,448.031,395.561,179.353,24.112,153.499
C07988=1097.317,447.785,395.604,179.352,24.099,153.496
C07989=1097.311,447.539,395.647,179.353,24.086,153.493
C07990=1097.304,447.293,395.691,179.352,24.074,153.489
C07991=1097.298,447.047,395.735,179.353,24.061,153.486
C07992=1097.291,446.801,395.779,179.352,24.048,153.483
C07993=1097.285,446.555,395.823,179.352,24.035,153.480
C07994=1097.279,446.309,395.867,179.351,24.023,153.477
C07995=1097.272,446.063,395.911,179.351,24.010,153.473
C07996=1097.267,445.817,395.954,179.349,23.996,153.470
C07997=1097.261,445.571,395.998,179.349,23.984,153.467
C07998=1097.254,445.325,396.041,179.347,23.971,153.464
C07999=1097.247,445.079,396.085,179.346,23.958,153.461
C08000=1097.241,444.833,396.128,179.344,23.945,153.458
C08001=1097.235,444.587,396.172,179.343,23.932,153.455
C08002=1097.229,444.341,396.215,179.341,23.919,153.452
C08003=1097.223,444.095,396.258,179.339,23.906,153.449
C08004=1097.216,443.849,396.302,179.337,23.893,153.446
C08005=1097.210,443.603,396.346,179.334,23.881,153.443
C08006=1097.204,443.356,396.389,179.332,23.868,153.440
C08007=1097.198,443.111,396.433,179.330,23.854,153.437
C08008=1097.192,442.864,396.476,179.327,23.842,153.434
C08009=1097.185,442.619,396.519,179.324,23.829,153.431
C08010=1097.179,442.373,396.562,179.323,23.816,153.428
C08011=1097.173,442.127,396.606,179.320,23.803,153.425
C08012=1097.167,441.880,396.649,179.318,23.791,153.422
C08013=1097.160,441.634,396.691,179.315,23.778,153.420
C08014=1097.154,441.389,396.735,179.312,23.766,153.417
C08015=1097.148,441.142,396.778,179.311,23.753,153.414
C08016=1097.142,440.896,396.821,179.308,23.741,153.411
C08017=1097.135,440.651,396.864,179.306,23.728,153.408
C08018=1097.129,440.404,396.907,179.303,23.716,153.405
C08019=1097.123,440.157,396.950,179.300,23.703,153.403
C08020=1097.117,439.912,396.993,179.299,23.691,153.400
C08021=1097.110,439.666,397.036,179.296,23.679,153.397
C08022=1097.104,439.420,397.079,179.293,23.667,153.394
C08023=1097.098,439.174,397.122,179.291,23.655,153.392
C08024=1097.092,438.927,397.165,179.289,23.643,153.389
C08025=1097.086,438.681,397.207,179.286,23.631,153.386
C08026=1097.080,438.435,397.250,179.284,23.619,153.384
C08027=1097.073,438.153,397.299,179.281,23.605,153.381
C08028=1097.065,437.870,397.348,179.278,23.591,153.378
C08029=1097.058,437.587,397.397,179.276,23.578,153.375
C08030=1097.051,437.305,397.446,179.272,23.564,153.372
C08031=1097.044,437.059,397.488,179.270,23.552,153.369
C08032=1097.039,436.813,397.531,179.268,23.541,153.366
C08033=1097.032,436.567,397.574,179.265,23.529,153.364
C08034=1097.026,436.321,397.617,179.263,23.518,153.361
C08035=1097.020,436.074,397.658,179.260,23.506,153.359
C08036=1097.014,435.828,397.701,179.257,23.494,153.356
C08037=1097.007,435.582,397.744,179.255,23.483,153.354
C08038=1097.002,435.336,397.786,179.253,23.471,153.351
C08039=1096.995,435.089,397.828,179.251,23.460,153.348
C08040=1096.990,434.843,397.871,179.248,23.449,153.346
C08041=1096.983,434.597,397.914,179.246,23.437,153.343
C08042=1096.977,434.351,397.955,179.243,23.426,153.341
C08043=1096.971,434.104,397.998,179.241,23.415,153.338
C08044=1096.964,433.858,398.040,179.238,23.403,153.336
C08045=1096.959,433.612,398.082,179.236,23.392,153.333
C08046=1096.952,433.366,398.125,179.233,23.381,153.331
C08047=1096.946,433.119,398.166,179.231,23.370,153.328
C08048=1096.940,432.873,398.210,179.228,23.359,153.326
C08049=1096.934,432.627,398.251,179.226,23.348,153.324
C08050=1096.928,432.380,398.294,179.223,23.337,153.321
C08051=1096.922,432.134,398.335,179.221,23.326,153.319
C08052=1096.916,431.888,398.376,179.218,23.315,153.317
C08053=1096.910,431.641,398.420,179.216,23.304,153.314
C08054=1096.904,431.395,398.461,179.213,23.293,153.312
C08055=1096.898,431.149,398.502,179.210,23.282,153.309
C08056=1096.891,430.903,398.545,179.208,23.272,153.307
C08057=1096.885,430.656,398.586,179.205,23.261,153.305
C08058=1096.879,430.410,398.628,179.203,23.250,153.303
C08059=1096.873,430.163,398.670,179.200,23.239,153.300
C08060=1096.867,429.917,398.713,179.198,23.229,153.298
C08061=1096.861,429.671,398.754,179.196,23.218,153.296
C08062=1096.854,429.424,398.796,179.192,23.208,153.293
C08063=1096.848,429.178,398.837,179.190,23.198,153.291
C08064=1096.842,428.932,398.879,179.188,23.187,153.289
C08065=1096.836,428.685,398.921,179.185,23.176,153.287
C08066=1096.830,428.439,398.962,179.183,23.166,153.284
C08067=1096.824,428.193,399.003,179.180,23.156,153.282
C08068=1096.817,427.946,399.045,179.177,23.145,153.280
C08069=1096.811,427.699,399.087,179.175,23.135,153.278
C08070=1096.806,427.453,399.128,179.172,23.125,153.276
C08071=1096.800,427.207,399.170,179.169,23.115,153.273
C08072=1096.793,426.960,399.211,179.167,23.104,153.271
C08073=1096.787,426.714,399.253,179.165,23.095,153.269
C08074=1096.781,426.468,399.294,179.162,23.085,153.267
C08075=1096.774,426.222,399.335,179.159,23.074,153.265
C08076=1096.768,425.974,399.376,179.157,23.064,153.263
C08077=1096.762,425.728,399.418,179.154,23.055,153.260
C08078=1096.756,425.482,399.459,179.152,23.045,153.258
C08079=1096.751,425.256,399.497,179.149,23.035,153.256
C08080=1096.746,425.030,399.535,179.147,23.026,153.255
C08081=1096.739,424.804,399.573,179.145,23.017,153.253
C08082=1096.734,424.578,399.611,179.142,23.008,153.251
C08083=1096.729,424.352,399.649,179.140,22.999,153.249
C08084=1096.723,424.127,399.686,179.137,22.990,153.247
C08085=1096.717,423.900,399.724,179.135,22.981,153.245
C08086=1096.712,423.674,399.761,179.132,22.972,153.243
C08087=1096.706,423.428,399.803,179.130,22.962,153.241
C08088=1096.700,423.182,399.844,179.128,22.953,153.239
C08089=1096.694,422.935,399.884,179.125,22.943,153.237
C08090=1096.688,422.689,399.926,179.123,22.934,153.235
C08091=1096.682,422.442,399.967,179.119,22.924,153.233
C08092=1096.675,422.195,400.008,179.117,22.915,153.231
C08093=1096.669,421.948,400.048,179.114,22.905,153.229
C08094=1096.664,421.702,400.089,179.112,22.896,153.227
C08095=1096.657,421.456,400.130,179.109,22.886,153.225
C08096=1096.652,421.209,400.171,179.107,22.877,153.223
C08097=1096.645,420.962,400.211,179.104,22.867,153.221
C08098=1096.639,420.716,400.252,179.101,22.859,153.219
C08099=1096.634,420.469,400.293,179.099,22.849,153.217
C08100=1096.627,420.223,400.333,179.096,22.840,153.216
C08101=1096.621,419.977,400.375,179.094,22.831,153.214
C08102=1096.615,419.730,400.415,179.091,22.822,153.212
C08103=1096.609,419.483,400.456,179.089,22.812,153.210
C08104=1096.604,419.237,400.496,179.086,22.803,153.208
C08105=1096.597,418.990,400.537,179.083,22.794,153.206
C08106=1096.591,418.744,400.578,179.081,22.785,153.204
C08107=1096.585,418.497,400.618,179.078,22.776,153.202
C08108=1096.579,418.250,400.659,179.075,22.767,153.200
C08109=1096.573,418.004,400.699,179.073,22.758,153.199
C08110=1096.567,417.757,400.740,179.070,22.749,153.197
C08111=1096.561,417.511,400.780,179.067,22.740,153.195
C08112=1096.555,417.264,400.821,179.065,22.731,153.193
C08113=1096.549,417.017,400.861,179.062,22.722,153.191
C08114=1096.543,416.770,400.902,179.060,22.713,153.189
C08115=1096.537,416.524,400.942,179.057,22.704,153.188
C08116=1096.531,416.277,400.982,179.054,22.695,153.186
C08117=1096.525,416.031,401.023,179.051,22.687,153.184
C08118=1096.519,415.783,401.062,179.049,22.678,153.182
C08119=1096.513,415.537,401.103,179.046,22.669,153.181
C08120=1096.507,415.290,401.143,179.044,22.661,153.179
C08121=1096.500,415.044,401.183,179.041,22.652,153.177
C08122=1096.494,414.797,401.223,179.038,22.644,153.175
C08123=1096.488,414.550,401.264,179.036,22.635,153.174
C08124=1096.482,414.303,401.303,179.033,22.626,153.172
C08125=1096.476,414.057,401.343,179.030,22.618,153.170
C08126=1096.470,413.811,401.383,179.027,22.609,153.168
C08127=1096.465,413.563,401.423,179.025,22.601,153.167
C08128=1096.458,413.317,401.464,179.022,22.593,153.165
C08129=1096.452,413.070,401.504,179.020,22.584,153.163
C08130=1096.446,412.823,401.543,179.017,22.576,153.162
C08131=1096.439,412.577,401.583,179.014,22.567,153.160
C08132=1096.434,412.329,401.623,179.012,22.559,153.158
C08133=1096.428,412.083,401.663,179.009,22.551,153.157
C08134=1096.422,411.837,401.703,179.006,22.543,153.155
C08135=1096.417,411.618,401.738,179.004,22.535,153.154
C08136=1096.411,411.399,401.774,179.002,22.528,153.152
C08137=1096.406,411.180,401.809,178.999,22.521,153.151
C08138=1096.401,410.961,401.845,178.997,22.514,153.149
C08139=1096.395,410.742,401.879,178.995,22.506,153.148
C08140=1096.390,410.523,401.915,178.993,22.499,153.146
C08141=1096.385,410.305,401.949,178.989,22.491,153.145
C08142=1096.379,410.086,401.985,178.987,22.484,153.144
C08143=1096.374,409.839,402.025,178.985,22.477,153.142
C08144=1096.368,409.591,402.064,178.982,22.468,153.140
C08145=1096.362,409.346,402.104,178.979,22.460,153.139
C08146=1096.356,409.098,402.144,178.977,22.452,153.137
C08147=1096.350,408.851,402.183,178.974,22.444,153.136
C08148=1096.344,408.605,402.223,178.971,22.436,153.134
C08149=1096.338,408.358,402.262,178.969,22.428,153.133
C08150=1096.332,408.111,402.302,178.966,22.420,153.131
C08151=1096.326,407.864,402.341,178.963,22.413,153.130
C08152=1096.321,407.618,402.380,178.961,22.405,153.128
C08153=1096.314,407.371,402.420,178.958,22.397,153.126
C08154=1096.308,407.124,402.460,178.955,22.389,153.125
C08155=1096.303,406.878,402.499,178.953,22.381,153.123
C08156=1096.297,406.630,402.538,178.950,22.373,153.122
C08157=1096.291,406.383,402.578,178.948,22.366,153.120
C08158=1096.285,406.137,402.617,178.945,22.358,153.119
C08159=1096.279,405.890,402.656,178.943,22.351,153.117
C08160=1096.273,405.643,402.696,178.939,22.343,153.116
C08161=1096.267,405.396,402.735,178.936,22.335,153.115
C08162=1096.261,405.149,402.774,178.934,22.327,153.113
C08163=1096.255,404.902,402.813,178.931,22.320,153.112
C08164=1096.249,404.656,402.852,178.929,22.312,153.110
C08165=1096.243,404.409,402.891,178.926,22.305,153.109
C08166=1096.238,404.162,402.931,178.924,22.297,153.107
C08167=1096.231,403.915,402.970,178.920,22.290,153.106
C08168=1096.225,403.668,403.009,178.918,22.283,153.104
C08169=1096.219,403.421,403.047,178.915,22.275,153.103
C08170=1096.213,403.174,403.087,178.913,22.268,153.102
C08171=1096.207,402.928,403.125,178.910,22.260,153.100
C08172=1096.201,402.681,403.165,178.907,22.253,153.099
C08173=1096.196,402.434,403.204,178.904,22.246,153.097
C08174=1096.190,402.187,403.242,178.902,22.238,153.096
C08175=1096.183,401.940,403.281,178.899,22.231,153.095
C08176=1096.178,401.693,403.320,178.896,22.224,153.093
C08177=1096.172,401.446,403.359,178.893,22.217,153.092
C08178=1096.166,401.199,403.397,178.891,22.209,153.090
C08179=1096.160,400.952,403.437,178.889,22.202,153.089
C08180=1096.154,400.705,403.475,178.885,22.195,153.088
C08181=1096.148,400.458,403.514,178.883,22.188,153.087
C08182=1096.142,400.212,403.553,178.880,22.180,153.085
C08183=1096.136,399.964,403.592,178.878,22.174,153.084
C08184=1096.130,399.718,403.630,178.874,22.166,153.082
C08185=1096.125,399.471,403.669,178.872,22.159,153.081
C08186=1096.118,399.224,403.707,178.870,22.152,153.080
C08187=1096.113,398.977,403.746,178.866,22.145,153.079
C08188=1096.106,398.730,403.785,178.864,22.138,153.077
C08189=1096.101,398.483,403.823,178.862,22.131,153.076
C08190=1096.094,398.237,403.862,178.858,22.124,153.075
C08191=1096.089,398.018,403.896,178.856,22.118,153.074
C08192=1096.084,397.799,403.929,178.854,22.112,153.072
C08193=1096.080,397.581,403.964,178.851,22.106,153.071
C08194=1096.074,397.362,403.998,178.849,22.100,153.070
C08195=1096.068,397.144,404.032,178.847,22.094,153.069
C08196=1096.064,396.924,404.066,178.844,22.088,153.068
C08197=1096.058,396.706,404.100,178.841,22.082,153.067
C08198=1096.053,396.487,404.134,178.839,22.075,153.066
C08199=1096.047,396.240,404.172,178.836,22.069,153.065
C08200=1096.041,395.994,404.210,178.834,22.062,153.063
C08201=1096.035,395.746,404.249,178.831,22.056,153.062
C08202=1096.029,395.500,404.287,178.828,22.049,153.061
C08203=1096.024,395.253,404.326,178.826,22.042,153.060
C08204=1096.017,395.005,404.364,178.823,22.035,153.058
C08205=1096.011,394.759,404.402,178.820,22.028,153.057
C08206=1096.005,394.512,404.440,178.817,22.022,153.056
C08207=1095.999,394.265,404.479,178.815,22.016,153.055
C08208=1095.994,394.018,404.516,178.812,22.009,153.054
C08209=1095.988,393.771,404.554,178.809,22.002,153.052
C08210=1095.982,393.524,404.592,178.806,21.996,153.051
C08211=1095.976,393.277,404.631,178.804,21.989,153.050
C08212=1095.970,393.030,404.668,178.801,21.983,153.049
C08213=1095.964,392.783,404.706,178.798,21.976,153.048
C08214=1095.959,392.536,404.744,178.795,21.969,153.047
C08215=1095.953,392.289,404.783,178.793,21.963,153.045
C08216=1095.947,392.042,404.820,178.790,21.957,153.044
C08217=1095.941,391.795,404.858,178.787,21.950,153.043
C08218=1095.935,391.548,404.896,178.784,21.944,153.042
C08219=1095.928,391.301,404.934,178.781,21.938,153.041
C08220=1095.922,391.054,404.972,178.779,21.931,153.040
C08221=1095.916,390.807,405.009,178.775,21.925,153.039
C08222=1095.911,390.561,405.047,178.773,21.918,153.038
C08223=1095.905,390.313,405.086,178.770,21.912,153.037
C08224=1095.899,390.066,405.124,178.767,21.906,153.035
C08225=1095.893,389.819,405.161,178.765,21.900,153.034
C08226=1095.887,389.572,405.198,178.761,21.893,153.033
C08227=1095.881,389.325,405.236,178.759,21.887,153.032
C08228=1095.876,389.079,405.274,178.756,21.881,153.031
C08229=1095.869,388.831,405.312,178.753,21.875,153.030
C08230=1095.863,388.584,405.350,178.751,21.869,153.029
C08231=1095.858,388.337,405.387,178.748,21.863,153.028
C08232=1095.852,388.090,405.425,178.744,21.856,153.027
C08233=1095.846,387.844,405.462,178.742,21.850,153.026
C08234=1095.839,387.596,405.499,178.739,21.844,153.025
C08235=1095.834,387.350,405.537,178.736,21.838,153.024
C08236=1095.828,387.103,405.574,178.734,21.831,153.023
C08237=1095.822,386.856,405.611,178.731,21.825,153.022
C08238=1095.816,386.609,405.649,178.727,21.819,153.021
C08239=1095.810,386.361,405.687,178.725,21.813,153.019
C08240=1095.804,386.114,405.724,178.722,21.807,153.018
C08241=1095.798,385.867,405.761,178.719,21.801,153.018
C08242=1095.793,385.620,405.799,178.716,21.795,153.016
C08243=1095.787,385.373,405.836,178.714,21.789,153.015
C08244=1095.781,385.126,405.874,178.711,21.783,153.014
C08245=1095.775,384.878,405.911,178.708,21.777,153.013
C08246=1095.770,384.632,405.949,178.705,21.771,153.012
C08247=1095.764,384.419,405.980,178.703,21.766,153.012
C08248=1095.759,384.208,406.012,178.700,21.761,153.011
C08249=1095.755,383.995,406.045,178.697,21.756,153.010
C08250=1095.749,383.783,406.076,178.695,21.751,153.009
C08251=1095.744,383.571,406.108,178.693,21.746,153.008
C08252=1095.740,383.359,406.140,178.690,21.740,153.007
C08253=1095.734,383.147,406.172,178.688,21.736,153.006
C08254=1095.729,382.934,406.204,178.686,21.731,153.006
C08255=1095.724,382.687,406.241,178.682,21.724,153.005
C08256=1095.718,382.440,406.278,178.679,21.719,153.004
C08257=1095.712,382.193,406.316,178.677,21.713,153.003
C08258=1095.706,381.946,406.352,178.674,21.707,153.002
C08259=1095.700,381.698,406.389,178.671,21.702,153.001
C08260=1095.694,381.451,406.426,178.668,21.696,153.000
C08261=1095.688,381.204,406.463,178.665,21.690,152.999
C08262=1095.682,380.957,406.501,178.662,21.685,152.998
C08263=1095.676,380.710,406.537,178.659,21.679,152.997
C08264=1095.670,380.463,406.574,178.657,21.674,152.996
C08265=1095.665,380.215,406.611,178.654,21.668,152.995
C08266=1095.659,379.969,406.647,178.651,21.662,152.995
C08267=1095.653,379.722,406.684,178.648,21.657,152.994
C08268=1095.647,379.475,406.721,178.645,21.651,152.993
C08269=1095.641,379.227,406.758,178.642,21.646,152.992
C08270=1095.636,378.980,406.795,178.639,21.640,152.991
C08271=1095.629,378.733,406.831,178.637,21.634,152.990
C08272=1095.624,378.486,406.868,178.634,21.629,152.989
C08273=1095.618,378.238,406.905,178.631,21.623,152.988
C08274=1095.612,377.991,406.942,178.628,21.618,152.987
C08275=1095.606,377.745,406.978,178.625,21.612,152.987
C08276=1095.601,377.497,407.015,178.622,21.607,152.986
C08277=1095.594,377.250,407.051,178.619,21.601,152.985
C08278=1095.589,377.003,407.088,178.616,21.596,152.984
C08279=1095.583,376.756,407.125,178.613,21.590,152.983
C08280=1095.577,376.509,407.162,178.610,21.585,152.982
C08281=1095.572,376.262,407.199,178.607,21.579,152.981
C08282=1095.566,376.014,407.234,178.604,21.574,152.980
C08283=1095.560,375.767,407.271,178.602,21.569,152.980
C08284=1095.554,375.520,407.308,178.599,21.563,152.979
C08285=1095.548,375.272,407.345,178.597,21.558,152.978
C08286=1095.543,375.025,407.380,178.594,21.553,152.977
C08287=1095.536,374.778,407.417,178.590,21.547,152.976
C08288=1095.531,374.531,407.454,178.588,21.542,152.975
C08289=1095.524,374.284,407.490,178.585,21.537,152.975
C08290=1095.520,374.037,407.526,178.582,21.531,152.974
C08291=1095.513,373.790,407.562,178.579,21.526,152.973
C08292=1095.507,373.542,407.598,178.576,21.521,152.972
C08293=1095.502,373.295,407.635,178.573,21.515,152.972
C08294=1095.495,373.048,407.672,178.570,21.510,152.971
C08295=1095.490,372.801,407.707,178.567,21.506,152.970
C08296=1095.484,372.554,407.744,178.564,21.500,152.969
C08297=1095.478,372.306,407.780,178.561,21.495,152.968
C08298=1095.472,372.059,407.816,178.558,21.490,152.968
C08299=1095.467,371.812,407.852,178.555,21.484,152.967
C08300=1095.460,371.564,407.888,178.552,21.479,152.966
C08301=1095.455,371.316,407.924,178.549,21.474,152.965
C08302=1095.449,371.069,407.961,178.546,21.469,152.965
C08303=1095.440,370.673,408.019,178.542,21.461,152.963
C08304=1095.430,370.275,408.077,178.537,21.453,152.962
C08305=1095.420,369.878,408.134,178.532,21.445,152.961
C08306=1095.411,369.481,408.192,178.527,21.437,152.960
C08307=1095.406,369.234,408.228,178.524,21.431,152.959
C08308=1095.400,368.987,408.264,178.522,21.427,152.958
C08309=1095.394,368.739,408.300,178.519,21.422,152.958
C08310=1095.388,368.492,408.335,178.516,21.417,152.957
C08311=1095.382,368.245,408.372,178.513,21.412,152.956
C08312=1095.376,367.997,408.407,178.510,21.406,152.955
C08313=1095.371,367.750,408.443,178.507,21.402,152.955
C08314=1095.365,367.502,408.479,178.504,21.397,152.954
C08315=1095.360,367.255,408.514,178.501,21.392,152.953
C08316=1095.354,367.008,408.551,178.498,21.387,152.952
C08317=1095.348,366.760,408.587,178.495,21.382,152.952
C08318=1095.342,366.514,408.622,178.492,21.377,152.951
C08319=1095.336,366.266,408.658,178.490,21.372,152.950
C08320=1095.331,366.019,408.693,178.486,21.368,152.950
C08321=1095.325,365.771,408.729,178.483,21.362,152.949
C08322=1095.319,365.524,408.764,178.480,21.358,152.948
C08323=1095.313,365.277,408.800,178.477,21.353,152.948
C08324=1095.307,365.029,408.836,178.475,21.348,152.947
C08325=1095.302,364.782,408.871,178.472,21.343,152.946
C08326=1095.296,364.534,408.907,178.468,21.339,152.946
C08327=1095.290,364.287,408.942,178.465,21.334,152.945
C08328=1095.284,364.040,408.978,178.463,21.329,152.944
C08329=1095.278,363.792,409.014,178.460,21.324,152.944
C08330=1095.273,363.545,409.049,178.457,21.320,152.943
C08331=1095.267,363.297,409.085,178.453,21.315,152.942
C08332=1095.261,363.051,409.119,178.451,21.311,152.942
C08333=1095.255,362.803,409.155,178.448,21.306,152.941
C08334=1095.249,362.556,409.191,178.444,21.301,152.941
C08335=1095.243,362.308,409.226,178.441,21.296,152.940
C08336=1095.238,362.061,409.261,178.439,21.292,152.939
C08337=1095.232,361.813,409.297,178.436,21.287,152.938
C08338=1095.226,361.566,409.332,178.433,21.282,152.938
C08339=1095.220,361.319,409.367,178.429,21.277,152.937
C08340=1095.215,361.071,409.402,178.427,21.273,152.937
C08341=1095.209,360.823,409.438,178.424,21.269,152.936
C08342=1095.203,360.576,409.473,178.420,21.264,152.935
C08343=1095.197,360.329,409.509,178.417,21.259,152.935
C08344=1095.191,360.081,409.543,178.415,21.255,152.934
C08345=1095.185,359.834,409.578,178.412,21.250,152.934
C08346=1095.180,359.587,409.614,178.408,21.245,152.933
C08347=1095.174,359.338,409.649,178.406,21.241,152.932
C08348=1095.168,359.092,409.684,178.403,21.237,152.932
C08349=1095.162,358.844,409.719,178.399,21.232,152.931
C08350=1095.157,358.597,409.754,178.397,21.228,152.931
C08351=1095.150,358.349,409.789,178.394,21.223,152.930
C08352=1095.145,358.102,409.824,178.390,21.218,152.930
C08353=1095.139,357.854,409.859,178.388,21.214,152.929
C08354=1095.133,357.607,409.893,178.385,21.210,152.928
C08355=1095.124,357.225,409.948,178.380,21.203,152.928
C08356=1095.115,356.843,410.001,178.375,21.196,152.927
C08357=1095.106,356.461,410.055,178.370,21.189,152.926
C08358=1095.097,356.079,410.109,178.366,21.183,152.925
C08359=1095.092,355.832,410.144,178.363,21.178,152.924
C08360=1095.086,355.583,410.179,178.360,21.174,152.924
C08361=1095.080,355.337,410.214,178.357,21.169,152.923
C08362=1095.075,355.089,410.248,178.353,21.165,152.923
C08363=1095.068,354.841,410.283,178.351,21.160,152.922
C08364=1095.063,354.594,410.318,178.348,21.156,152.922
C08365=1095.057,354.347,410.352,178.344,21.152,152.921
C08366=1095.051,354.098,410.387,178.342,21.148,152.920
C08367=1095.046,353.851,410.423,178.338,21.143,152.920
C08368=1095.040,353.604,410.457,178.336,21.139,152.919
C08369=1095.034,353.356,410.492,178.333,21.135,152.919
C08370=1095.028,353.109,410.526,178.329,21.130,152.918
C08371=1095.023,352.861,410.560,178.327,21.126,152.918
C08372=1095.016,352.614,410.596,178.323,21.122,152.917
C08373=1095.011,352.366,410.630,178.321,21.118,152.917
C08374=1095.005,352.119,410.664,178.318,21.113,152.916
C08375=1094.999,351.871,410.699,178.314,21.109,152.916
C08376=1094.993,351.623,410.733,178.312,21.105,152.915
C08377=1094.988,351.376,410.767,178.308,21.101,152.915
C08378=1094.982,351.129,410.801,178.306,21.097,152.914
C08379=1094.976,350.880,410.836,178.302,21.093,152.914
C08380=1094.971,350.633,410.870,178.299,21.088,152.913
C08381=1094.965,350.386,410.905,178.296,21.084,152.913
C08382=1094.959,350.137,410.940,178.293,21.080,152.912
C08383=1094.953,349.890,410.974,178.290,21.076,152.912
C08384=1094.947,349.643,411.008,178.287,21.072,152.911
C08385=1094.942,349.395,411.042,178.283,21.068,152.911
C08386=1094.936,349.147,411.077,178.281,21.064,152.910
C08387=1094.930,348.900,411.111,178.277,21.059,152.910
C08388=1094.925,348.652,411.145,178.275,21.056,152.909
C08389=1094.919,348.405,411.179,178.272,21.051,152.909
C08390=1094.913,348.158,411.214,178.269,21.047,152.909
C08391=1094.907,347.910,411.248,178.266,21.043,152.908
C08392=1094.901,347.662,411.283,178.263,21.039,152.908
C08393=1094.896,347.415,411.317,178.259,21.035,152.907
C08394=1094.890,347.167,411.350,178.256,21.031,152.907
C08395=1094.884,346.920,411.384,178.253,21.027,152.906
C08396=1094.878,346.672,411.419,178.250,21.023,152.906
C08397=1094.873,346.424,411.453,178.248,21.019,152.905
C08398=1094.867,346.176,411.486,178.244,21.015,152.905
C08399=1094.861,345.929,411.520,178.241,21.011,152.904
C08400=1094.855,345.682,411.555,178.238,21.007,152.904
C08401=1094.850,345.434,411.589,178.235,21.003,152.903
C08402=1094.845,345.186,411.623,178.232,20.999,152.903
C08403=1094.838,344.938,411.657,178.229,20.995,152.903
C08404=1094.832,344.691,411.691,178.226,20.991,152.902
C08405=1094.827,344.443,411.724,178.223,20.987,152.902
C08406=1094.821,344.196,411.758,178.219,20.983,152.901
C08407=1094.812,343.816,411.810,178.215,20.977,152.901
C08408=1094.803,343.437,411.862,178.210,20.971,152.900
C08409=1094.794,343.058,411.914,178.205,20.965,152.899
C08410=1094.785,342.677,411.965,178.201,20.960,152.899
C08411=1094.779,342.430,411.999,178.198,20.956,152.898
C08412=1094.774,342.182,412.032,178.195,20.952,152.898
C08413=1094.768,341.935,412.066,178.191,20.948,152.898
C08414=1094.762,341.687,412.100,178.189,20.944,152.897
C08415=1094.756,341.440,412.134,178.185,20.940,152.897
C08416=1094.751,341.192,412.167,178.183,20.937,152.896
C08417=1094.745,340.944,412.201,178.179,20.932,152.896
C08418=1094.739,340.697,412.235,178.176,20.929,152.896
C08419=1094.734,340.449,412.268,178.173,20.925,152.895
C08420=1094.728,340.201,412.302,178.170,20.921,152.895
C08421=1094.722,339.953,412.336,178.167,20.917,152.894
C08422=1094.716,339.705,412.369,178.164,20.914,152.894
C08423=1094.710,339.458,412.403,178.161,20.909,152.894
C08424=1094.705,339.210,412.436,178.158,20.906,152.893
C08425=1094.699,338.962,412.470,178.155,20.903,152.893
C08426=1094.694,338.714,412.503,178.152,20.898,152.892
C08427=1094.688,338.467,412.537,178.149,20.895,152.892
C08428=1094.682,338.219,412.570,178.145,20.891,152.892
C08429=1094.676,337.971,412.603,178.143,20.888,152.891
C08430=1094.671,337.723,412.637,178.139,20.884,152.891
C08431=1094.665,337.476,412.671,178.136,20.880,152.891
C08432=1094.659,337.228,412.704,178.133,20.877,152.890
C08433=1094.653,336.980,412.737,178.130,20.873,152.890
C08434=1094.647,336.732,412.770,178.127,20.869,152.890
C08435=1094.642,336.485,412.803,178.124,20.866,152.889
C08436=1094.636,336.237,412.837,178.121,20.862,152.889
C08437=1094.631,335.990,412.869,178.118,20.858,152.889
C08438=1094.625,335.742,412.902,178.115,20.854,152.888
C08439=1094.619,335.494,412.936,178.112,20.851,152.888
C08440=1094.613,335.246,412.969,178.108,20.847,152.888
C08441=1094.608,334.998,413.002,178.106,20.844,152.887
C08442=1094.602,334.751,413.035,178.103,20.841,152.887
C08443=1094.596,334.503,413.069,178.099,20.837,152.887
C08444=1094.590,334.255,413.101,178.096,20.833,152.886
C08445=1094.585,334.007,413.135,178.093,20.829,152.886
C08446=1094.579,333.759,413.168,178.090,20.826,152.886
C08447=1094.573,333.512,413.201,178.087,20.823,152.885
C08448=1094.567,333.264,413.234,178.084,20.819,152.885
C08449=1094.562,333.017,413.267,178.081,20.815,152.885
C08450=1094.556,332.769,413.300,178.078,20.812,152.884
C08451=1094.550,332.521,413.333,178.074,20.808,152.884
C08452=1094.545,332.273,413.366,178.072,20.804,152.884
C08453=1094.539,332.026,413.399,178.068,20.800,152.883
C08454=1094.533,331.777,413.432,178.065,20.798,152.883
C08455=1094.527,331.529,413.465,178.062,20.794,152.883
C08456=1094.521,331.282,413.497,178.059,20.791,152.882
C08457=1094.516,331.035,413.530,178.056,20.787,152.882
C08458=1094.509,330.787,413.563,178.053,20.784,152.882
C08459=1094.501,330.401,413.614,178.048,20.778,152.881
C08460=1094.492,330.016,413.665,178.043,20.773,152.881
C08461=1094.482,329.630,413.716,178.039,20.768,152.880
C08462=1094.473,329.245,413.766,178.034,20.763,152.880
C08463=1094.468,328.996,413.799,178.030,20.759,152.880
C08464=1094.462,328.749,413.832,178.027,20.756,152.879
C08465=1094.456,328.501,413.865,178.024,20.753,152.879
C08466=1094.450,328.253,413.897,178.021,20.749,152.879
C08467=1094.444,328.006,413.929,178.018,20.746,152.879
C08468=1094.439,327.758,413.963,178.015,20.742,152.878
C08469=1094.433,327.510,413.995,178.012,20.739,152.878
C08470=1094.426,327.262,414.028,178.008,20.735,152.878
C08471=1094.421,327.014,414.060,178.005,20.733,152.878
C08472=1094.416,326.767,414.093,178.003,20.729,152.877
C08473=1094.410,326.518,414.125,177.999,20.726,152.877
C08474=1094.403,326.271,414.157,177.996,20.722,152.877
C08475=1094.398,326.022,414.190,177.993,20.719,152.877
C08476=1094.392,325.775,414.222,177.990,20.716,152.876
C08477=1094.386,325.527,414.254,177.987,20.712,152.876
C08478=1094.381,325.279,414.287,177.984,20.709,152.876
C08479=1094.375,325.031,414.320,177.981,20.706,152.875
C08480=1094.369,324.784,414.351,177.977,20.702,152.875
C08481=1094.363,324.536,414.384,177.974,20.699,152.875
C08482=1094.358,324.287,414.417,177.971,20.696,152.875
C08483=1094.352,324.040,414.448,177.968,20.693,152.875
C08484=1094.346,323.792,414.481,177.965,20.689,152.874
C08485=1094.340,323.544,414.513,177.962,20.686,152.874
C08486=1094.336,323.296,414.545,177.959,20.683,152.874
C08487=1094.329,323.049,414.578,177.956,20.680,152.873
C08488=1094.323,322.800,414.610,177.952,20.676,152.873
C08489=1094.318,322.553,414.642,177.950,20.673,152.873
C08490=1094.312,322.305,414.674,177.947,20.670,152.873
C08491=1094.306,322.057,414.707,177.944,20.667,152.873
C08492=1094.301,321.809,414.739,177.940,20.663,152.872
C08493=1094.295,321.561,414.771,177.937,20.660,152.872
C08494=1094.290,321.314,414.803,177.934,20.657,152.872
C08495=1094.284,321.065,414.835,177.931,20.654,152.872
C08496=1094.277,320.818,414.867,177.928,20.650,152.871
C08497=1094.273,320.570,414.900,177.925,20.647,152.871
C08498=1094.267,320.322,414.932,177.922,20.644,152.871
C08499=1094.261,320.074,414.963,177.919,20.641,152.871
C08500=1094.255,319.826,414.995,177.915,20.638,152.870
C08501=1094.250,319.579,415.027,177.912,20.634,152.870
C08502=1094.244,319.330,415.059,177.909,20.631,152.870
C08503=1094.239,319.083,415.091,177.907,20.628,152.870
C08504=1094.233,318.834,415.123,177.904,20.625,152.870
C08505=1094.228,318.587,415.155,177.900,20.622,152.869
C08506=1094.222,318.339,415.187,177.897,20.618,152.869
C08507=1094.217,318.091,415.219,177.894,20.615,152.869
C08508=1094.211,317.843,415.251,177.891,20.612,152.869
C08509=1094.205,317.595,415.282,177.888,20.609,152.868
C08510=1094.199,317.347,415.314,177.884,20.606,152.868
C08511=1094.190,316.955,415.365,177.880,20.601,152.868
C08512=1094.182,316.562,415.415,177.875,20.596,152.867
C08513=1094.173,316.170,415.465,177.870,20.590,152.867
C08514=1094.164,315.778,415.515,177.865,20.586,152.867
C08515=1094.158,315.529,415.548,177.863,20.583,152.867
C08516=1094.153,315.281,415.578,177.859,20.580,152.866
C08517=1094.147,315.034,415.610,177.856,20.577,152.866
C08518=1094.141,314.786,415.642,177.853,20.574,152.866
C08519=1094.135,314.537,415.674,177.850,20.571,152.866
C08520=1094.130,314.290,415.706,177.847,20.568,152.866
C08521=1094.124,314.041,415.737,177.844,20.565,152.866
C08522=1094.118,313.794,415.768,177.840,20.562,152.865
C08523=1094.112,313.546,415.800,177.837,20.559,152.865
C08524=1094.106,313.298,415.831,177.834,20.556,152.865
C08525=1094.100,313.050,415.863,177.831,20.553,152.865
C08526=1094.095,312.802,415.894,177.828,20.550,152.865
C08527=1094.089,312.555,415.925,177.825,20.547,152.864
C08528=1094.083,312.306,415.957,177.821,20.544,152.864
C08529=1094.078,312.059,415.988,177.818,20.541,152.864
C08530=1094.071,311.811,416.020,177.815,20.538,152.864
C08531=1094.066,311.563,416.051,177.812,20.535,152.864
C08532=1094.060,311.314,416.083,177.809,20.532,152.864
C08533=1094.054,311.066,416.113,177.806,20.530,152.864
C08534=1094.049,310.819,416.145,177.803,20.527,152.863
C08535=1094.043,310.570,416.176,177.799,20.523,152.863
C08536=1094.037,310.323,416.207,177.796,20.521,152.863
C08537=1094.031,310.075,416.239,177.793,20.518,152.863
C08538=1094.025,309.827,416.269,177.790,20.515,152.863
C08539=1094.020,309.579,416.301,177.787,20.512,152.863
C08540=1094.014,309.331,416.332,177.784,20.509,152.862
C08541=1094.008,309.083,416.364,177.781,20.506,152.862
C08542=1094.003,308.835,416.394,177.777,20.503,152.862
C08543=1093.996,308.587,416.425,177.774,20.500,152.862
C08544=1093.991,308.339,416.457,177.771,20.497,152.862
C08545=1093.985,308.091,416.487,177.768,20.495,152.862
C08546=1093.979,307.843,416.519,177.765,20.492,152.862
C08547=1093.973,307.595,416.550,177.762,20.489,152.861
C08548=1093.968,307.347,416.581,177.759,20.486,152.861
C08549=1093.963,307.100,416.612,177.756,20.483,152.861
C08550=1093.957,306.851,416.643,177.752,20.480,152.861
C08551=1093.952,306.603,416.674,177.749,20.477,152.861
C08552=1093.945,306.356,416.705,177.746,20.474,152.861
C08553=1093.940,306.107,416.736,177.743,20.471,152.861
C08554=1093.934,305.859,416.767,177.740,20.468,152.860
C08555=1093.929,305.612,416.798,177.737,20.465,152.860
C08556=1093.923,305.364,416.829,177.734,20.463,152.860
C08557=1093.918,305.116,416.860,177.731,20.460,152.860
C08558=1093.911,304.867,416.890,177.727,20.457,152.860
C08559=1093.906,304.620,416.922,177.724,20.454,152.860
C08560=1093.900,304.372,416.952,177.721,20.451,152.860
C08561=1093.895,304.124,416.983,177.718,20.448,152.860
C08562=1093.889,303.876,417.014,177.715,20.445,152.859
C08563=1093.880,303.486,417.062,177.711,20.441,152.859
C08564=1093.872,303.096,417.111,177.705,20.436,152.859
C08565=1093.862,302.706,417.159,177.701,20.432,152.859
C08566=1093.853,302.317,417.207,177.695,20.428,152.859
C08567=1093.848,302.069,417.238,177.692,20.425,152.858
C08568=1093.842,301.820,417.269,177.689,20.422,152.858
C08569=1093.836,301.572,417.299,177.686,20.419,152.858
C08570=1093.831,301.324,417.330,177.683,20.416,152.858
C08571=1093.825,301.076,417.360,177.680,20.414,152.858
C08572=1093.820,300.828,417.391,177.677,20.411,152.858
C08573=1093.814,300.580,417.422,177.674,20.408,152.858
C08574=1093.809,300.333,417.452,177.671,20.405,152.858
C08575=1093.803,300.084,417.483,177.668,20.403,152.857
C08576=1093.798,299.837,417.513,177.665,20.400,152.857
C08577=1093.792,299.589,417.544,177.661,20.397,152.857
C08578=1093.787,299.341,417.575,177.658,20.394,152.857
C08579=1093.781,299.092,417.604,177.655,20.391,152.857
C08580=1093.775,298.844,417.635,177.652,20.388,152.857
C08581=1093.770,298.596,417.665,177.649,20.386,152.857
C08582=1093.765,298.348,417.696,177.646,20.383,152.857
C08583=1093.759,298.101,417.726,177.643,20.380,152.857
C08584=1093.753,297.852,417.757,177.640,20.377,152.856
C08585=1093.748,297.603,417.787,177.636,20.375,152.856
C08586=1093.742,297.355,417.817,177.633,20.372,152.856
C08587=1093.736,297.108,417.848,177.630,20.369,152.856
C08588=1093.730,296.860,417.878,177.627,20.367,152.856
C08589=1093.725,296.611,417.908,177.624,20.364,152.856
C08590=1093.719,296.364,417.938,177.621,20.361,152.856
C08591=1093.714,296.115,417.969,177.618,20.359,152.856
C08592=1093.708,295.868,417.999,177.615,20.356,152.856
C08593=1093.702,295.619,418.029,177.612,20.353,152.856
C08594=1093.697,295.371,418.059,177.609,20.351,152.856
C08595=1093.691,295.124,418.090,177.605,20.348,152.855
C08596=1093.685,294.875,418.119,177.602,20.346,152.855
C08597=1093.679,294.627,418.150,177.599,20.343,152.855
C08598=1093.674,294.379,418.179,177.596,20.340,152.855
C08599=1093.668,294.131,418.210,177.593,20.338,152.855
C08600=1093.662,293.883,418.240,177.590,20.335,152.855
C08601=1093.657,293.635,418.270,177.587,20.332,152.855
C08602=1093.651,293.387,418.300,177.584,20.330,152.855
C08603=1093.645,293.139,418.330,177.581,20.327,152.855
C08604=1093.640,292.891,418.360,177.578,20.324,152.855
C08605=1093.634,292.642,418.390,177.574,20.322,152.855
C08606=1093.628,292.394,418.420,177.571,20.319,152.855
C08607=1093.623,292.146,418.450,177.568,20.317,152.855
C08608=1093.617,291.898,418.480,177.565,20.314,152.855
C08609=1093.611,291.650,418.510,177.562,20.311,152.854
C08610=1093.606,291.402,418.540,177.559,20.309,152.854
C08611=1093.600,291.153,418.570,177.556,20.306,152.854
C08612=1093.594,290.905,418.599,177.553,20.304,152.854
C08613=1093.588,290.657,418.629,177.549,20.301,152.854
C08614=1093.582,290.409,418.659,177.546,20.299,152.854
C08615=1093.574,290.033,418.704,177.542,20.295,152.854
C08616=1093.566,289.657,418.749,177.537,20.290,152.854
C08617=1093.558,289.282,418.794,177.532,20.287,152.854
C08618=1093.549,288.906,418.839,177.527,20.283,152.854
C08619=1093.543,288.657,418.868,177.524,20.280,152.854
C08620=1093.537,288.410,418.898,177.521,20.278,152.854
C08621=1093.531,288.162,418.928,177.518,20.275,152.854
C08622=1093.526,287.913,418.958,177.515,20.273,152.854
C08623=1093.520,287.665,418.987,177.512,20.270,152.853
C08624=1093.514,287.417,419.017,177.509,20.268,152.853
C08625=1093.508,287.169,419.047,177.505,20.265,152.853
C08626=1093.503,286.920,419.076,177.502,20.263,152.853
C08627=1093.497,286.672,419.105,177.499,20.260,152.853
C08628=1093.492,286.424,419.134,177.496,20.257,152.853
C08629=1093.486,286.176,419.164,177.493,20.255,152.853
C08630=1093.480,285.928,419.194,177.490,20.252,152.853
C08631=1093.474,285.680,419.224,177.487,20.250,152.853
C08632=1093.469,285.432,419.253,177.483,20.248,152.853
C08633=1093.463,285.183,419.283,177.480,20.245,152.853
C08634=1093.457,284.936,419.311,177.477,20.243,152.853
C08635=1093.452,284.687,419.341,177.475,20.241,152.853
C08636=1093.446,284.439,419.371,177.471,20.238,152.853
C08637=1093.440,284.191,419.400,177.468,20.236,152.853
C08638=1093.435,283.942,419.429,177.465,20.233,152.853
C08639=1093.430,283.694,419.459,177.462,20.230,152.853
C08640=1093.423,283.446,419.488,177.459,20.228,152.853
C08641=1093.418,283.198,419.517,177.456,20.225,152.853
C08642=1093.412,282.949,419.547,177.452,20.223,152.853
C08643=1093.407,282.702,419.576,177.449,20.220,152.853
C08644=1093.401,282.454,419.605,177.446,20.218,152.853
C08645=1093.395,282.205,419.634,177.443,20.215,152.853
C08646=1093.389,281.957,419.664,177.440,20.213,152.853
C08647=1093.385,281.709,419.693,177.437,20.210,152.852
C08648=1093.379,281.461,419.722,177.434,20.208,152.852
C08649=1093.373,281.212,419.751,177.431,20.206,152.852
C08650=1093.367,280.964,419.780,177.428,20.203,152.852
C08651=1093.362,280.716,419.810,177.425,20.201,152.852
C08652=1093.356,280.468,419.839,177.422,20.198,152.852
C08653=1093.351,280.219,419.867,177.418,20.196,152.852
C08654=1093.344,279.971,419.897,177.415,20.193,152.852
C08655=1093.339,279.723,419.926,177.412,20.191,152.852
C08656=1093.333,279.475,419.955,177.409,20.189,152.852
C08657=1093.328,279.226,419.984,177.406,20.186,152.852
C08658=1093.322,278.979,420.012,177.402,20.184,152.852
C08659=1093.316,278.730,420.041,177.400,20.182,152.852
C08660=1093.311,278.481,420.070,177.397,20.179,152.852
C08661=1093.305,278.234,420.099,177.394,20.176,152.852
C08662=1093.300,277.985,420.129,177.390,20.174,152.852
C08663=1093.294,277.737,420.157,177.387,20.172,152.852
C08664=1093.289,277.489,420.186,177.384,20.169,152.852
C08665=1093.283,277.241,420.215,177.381,20.167,152.852
C08666=1093.277,276.992,420.244,177.378,20.164,152.852
C08667=1093.269,276.626,420.286,177.374,20.161,152.852
C08668=1093.260,276.259,420.329,177.369,20.157,152.852
C08669=1093.252,275.893,420.371,177.364,20.154,152.852
C08670=1093.244,275.526,420.414,177.359,20.150,152.852
C08671=1093.238,275.278,420.443,177.357,20.148,152.852
C08672=1093.232,275.030,420.471,177.354,20.146,152.852
C08673=1093.227,274.782,420.500,177.351,20.144,152.852
C08674=1093.221,274.533,420.529,177.347,20.141,152.852
C08675=1093.215,274.285,420.558,177.344,20.139,152.852
C08676=1093.210,274.037,420.586,177.341,20.136,152.852
C08677=1093.204,273.788,420.615,177.338,20.134,152.852
C08678=1093.199,273.540,420.643,177.335,20.132,152.852
C08679=1093.193,273.292,420.672,177.332,20.129,152.852
C08680=1093.186,273.043,420.701,177.329,20.127,152.852
C08681=1093.182,272.795,420.729,177.326,20.125,152.852
C08682=1093.176,272.547,420.758,177.323,20.122,152.852
C08683=1093.170,272.299,420.786,177.319,20.120,152.852
C08684=1093.164,272.050,420.815,177.316,20.118,152.852
C08685=1093.159,271.803,420.843,177.314,20.116,152.852
C08686=1093.153,271.554,420.872,177.310,20.113,152.852
C08687=1093.148,271.305,420.900,177.307,20.111,152.852
C08688=1093.142,271.057,420.928,177.304,20.108,152.852
C08689=1093.136,270.809,420.957,177.301,20.106,152.852
C08690=1093.131,270.561,420.985,177.298,20.104,152.852
C08691=1093.125,270.312,421.014,177.295,20.102,152.852
C08692=1093.119,270.064,421.042,177.292,20.100,152.852
C08693=1093.113,269.816,421.071,177.289,20.097,152.852
C08694=1093.108,269.568,421.099,177.286,20.094,152.852
C08695=1093.102,269.319,421.127,177.282,20.092,152.852
C08696=1093.096,269.071,421.155,177.279,20.090,152.852
C08697=1093.091,268.822,421.184,177.277,20.088,152.852
C08698=1093.086,268.574,421.212,177.273,20.086,152.852
C08699=1093.080,268.326,421.241,177.270,20.083,152.852
C08700=1093.074,268.078,421.269,177.267,20.081,152.852
C08701=1093.068,267.829,421.297,177.264,20.079,152.852
C08702=1093.063,267.581,421.325,177.261,20.077,152.852
C08703=1093.057,267.332,421.353,177.258,20.074,152.852
C08704=1093.052,267.084,421.381,177.255,20.072,152.852
C08705=1093.046,266.835,421.410,177.252,20.070,152.852
C08706=1093.040,266.587,421.438,177.248,20.067,152.852
C08707=1093.035,266.338,421.466,177.245,20.065,152.852
C08708=1093.029,266.090,421.494,177.243,20.063,152.852
C08709=1093.023,265.842,421.522,177.240,20.061,152.852
C08710=1093.017,265.594,421.550,177.236,20.059,152.852
C08711=1093.012,265.346,421.578,177.233,20.056,152.852
C08712=1093.006,265.097,421.606,177.230,20.054,152.852
C08713=1093.001,264.849,421.634,177.227,20.052,152.852
C08714=1092.995,264.600,421.662,177.224,20.050,152.852
C08715=1092.989,264.352,421.690,177.221,20.047,152.852
C08716=1092.984,264.103,421.718,177.217,20.045,152.853
C08717=1092.978,263.855,421.746,177.214,20.043,152.852
C08718=1092.972,263.606,421.774,177.212,20.041,152.853
C08719=1092.964,263.244,421.814,177.207,20.037,152.853
C08720=1092.955,262.879,421.855,177.203,20.034,152.853
C08721=1092.947,262.516,421.896,177.198,20.031,152.853
C08722=1092.939,262.152,421.937,177.194,20.028,152.853
C08723=1092.933,261.904,421.964,177.191,20.026,152.853
C08724=1092.927,261.655,421.992,177.187,20.024,152.853
C08725=1092.921,261.407,422.020,177.184,20.021,152.853
C08726=1092.916,261.158,422.048,177.181,20.019,152.853
C08727=1092.910,260.910,422.075,177.178,20.017,152.853
C08728=1092.904,260.662,422.103,177.175,20.015,152.853
C08729=1092.899,260.413,422.131,177.172,20.013,152.853
C08730=1092.892,260.165,422.158,177.168,20.011,152.853
C08731=1092.887,259.916,422.187,177.166,20.009,152.853
C08732=1092.881,259.668,422.213,177.163,20.006,152.853
C08733=1092.875,259.420,422.241,177.159,20.004,152.853
C08734=1092.869,259.171,422.269,177.156,20.002,152.853
C08735=1092.864,258.923,422.296,177.154,20.000,152.853
C08736=1092.858,258.674,422.324,177.151,19.998,152.853
C08737=1092.853,258.425,422.352,177.147,19.996,152.853
C08738=1092.847,258.177,422.379,177.144,19.994,152.854
C08739=1092.841,257.929,422.407,177.142,19.992,152.853
C08740=1092.835,257.680,422.434,177.138,19.989,152.854
C08741=1092.830,257.432,422.462,177.135,19.987,152.854
C08742=1092.825,257.184,422.489,177.132,19.985,152.854
C08743=1092.818,256.936,422.517,177.129,19.983,152.854
C08744=1092.813,256.686,422.544,177.126,19.981,152.854
C08745=1092.807,256.439,422.572,177.123,19.979,152.854
C08746=1092.802,256.190,422.599,177.119,19.976,152.854
C08747=1092.796,255.941,422.626,177.117,19.974,152.854
C08748=1092.790,255.693,422.654,177.114,19.972,152.854
C08749=1092.785,255.444,422.681,177.110,19.970,152.854
C08750=1092.779,255.196,422.708,177.107,19.968,152.854
C08751=1092.773,254.947,422.736,177.105,19.966,152.854
C08752=1092.767,254.699,422.763,177.101,19.964,152.854
C08753=1092.762,254.451,422.791,177.098,19.961,152.854
C08754=1092.756,254.202,422.817,177.095,19.959,152.854
C08755=1092.751,253.954,422.845,177.093,19.957,152.854
C08756=1092.745,253.705,422.872,177.089,19.955,152.854
C08757=1092.740,253.457,422.899,177.086,19.953,152.854
C08758=1092.734,253.208,422.926,177.084,19.951,152.854
C08759=1092.728,252.960,422.954,177.080,19.949,152.854
C08760=1092.723,252.712,422.981,177.077,19.946,152.854
C08761=1092.718,252.463,423.008,177.074,19.944,152.855
C08762=1092.711,252.214,423.035,177.071,19.942,152.854
C08763=1092.706,251.966,423.063,177.068,19.940,152.855
C08764=1092.700,251.718,423.090,177.065,19.938,152.855
C08765=1092.695,251.469,423.117,177.062,19.936,152.855
C08766=1092.689,251.221,423.143,177.059,19.934,152.855
C08767=1092.684,250.972,423.171,177.056,19.931,152.855
C08768=1092.678,250.724,423.198,177.052,19.929,152.855
C08769=1092.673,250.476,423.225,177.050,19.927,152.855
C08770=1092.667,250.226,423.252,177.047,19.925,152.855
C08771=1092.659,249.860,423.292,177.043,19.922,152.855
C08772=1092.651,249.494,423.332,177.038,19.919,152.855
C08773=1092.642,249.127,423.372,177.034,19.916,152.855
C08774=1092.635,248.761,423.412,177.029,19.912,152.855
C08775=1092.629,248.512,423.438,177.026,19.910,152.855
C08776=1092.624,248.263,423.466,177.023,19.908,152.855
C08777=1092.618,248.014,423.493,177.020,19.906,152.855
C08778=1092.612,247.766,423.519,177.016,19.904,152.855
C08779=1092.607,247.517,423.546,177.014,19.902,152.855
C08780=1092.601,247.269,423.573,177.011,19.900,152.855
C08781=1092.595,247.021,423.600,177.008,19.897,152.855
C08782=1092.590,246.772,423.627,177.005,19.896,152.855
C08783=1092.584,246.524,423.654,177.002,19.893,152.856
C08784=1092.579,246.275,423.680,176.999,19.891,152.856
C08785=1092.573,246.026,423.706,176.996,19.889,152.856
C08786=1092.568,245.778,423.734,176.993,19.887,152.856
C08787=1092.562,245.529,423.760,176.990,19.885,152.856
C08788=1092.557,245.281,423.787,176.987,19.883,152.856
C08789=1092.551,245.033,423.813,176.984,19.881,152.856
C08790=1092.545,244.784,423.840,176.981,19.879,152.856
C08791=1092.540,244.536,423.867,176.978,19.877,152.856
C08792=1092.535,244.287,423.893,176.975,19.875,152.856
C08793=1092.529,244.038,423.920,176.972,19.872,152.856
C08794=1092.523,243.790,423.947,176.969,19.871,152.856
C08795=1092.517,243.541,423.973,176.966,19.869,152.856
C08796=1092.512,243.292,423.999,176.962,19.866,152.856
C08797=1092.507,243.044,424.026,176.960,19.865,152.856
C08798=1092.501,242.795,424.053,176.957,19.862,152.857
C08799=1092.495,242.547,424.080,176.953,19.860,152.856
C08800=1092.490,242.298,424.106,176.951,19.858,152.857
C08801=1092.484,242.050,424.132,176.948,19.856,152.857
C08802=1092.478,241.801,424.159,176.944,19.854,152.857
C08803=1092.473,241.552,424.185,176.942,19.852,152.857
C08804=1092.467,241.304,424.211,176.939,19.850,152.857
C08805=1092.461,241.056,424.238,176.935,19.848,152.857
C08806=1092.456,240.807,424.264,176.933,19.846,152.857
C08807=1092.450,240.558,424.291,176.929,19.844,152.857
C08808=1092.444,240.310,424.317,176.926,19.842,152.857
C08809=1092.439,240.061,424.343,176.924,19.840,152.857
C08810=1092.433,239.813,424.370,176.920,19.838,152.857
C08811=1092.427,239.564,424.396,176.918,19.836,152.857
C08812=1092.422,239.315,424.423,176.915,19.834,152.857
C08813=1092.416,239.066,424.448,176.911,19.832,152.858
C08814=1092.410,238.818,424.475,176.909,19.830,152.858
C08815=1092.404,238.570,424.501,176.906,19.828,152.858
C08816=1092.399,238.322,424.527,176.902,19.826,152.858
C08817=1092.393,238.073,424.553,176.900,19.824,152.858
C08818=1092.388,237.824,424.579,176.896,19.822,152.858
C08819=1092.382,237.575,424.605,176.894,19.820,152.858
C08820=1092.377,237.327,424.632,176.891,19.818,152.858
C08821=1092.371,237.078,424.658,176.887,19.816,152.858
C08822=1092.365,236.830,424.684,176.885,19.814,152.858
C08823=1092.357,236.456,424.723,176.880,19.811,152.858
C08824=1092.349,236.083,424.762,176.876,19.808,152.858
C08825=1092.340,235.709,424.802,176.871,19.804,152.858
C08826=1092.332,235.336,424.841,176.867,19.802,152.859
C08827=1092.326,235.087,424.867,176.863,19.800,152.859
C08828=1092.321,234.838,424.893,176.861,19.798,152.859
C08829=1092.315,234.590,424.919,176.858,19.796,152.859
C08830=1092.309,234.341,424.945,176.855,19.794,152.859
C08831=1092.304,234.092,424.971,176.852,19.792,152.859
C08832=1092.298,233.844,424.997,176.849,19.789,152.859
C08833=1092.293,233.595,425.023,176.846,19.788,152.859
C08834=1092.287,233.347,425.048,176.843,19.786,152.859
C08835=1092.282,233.098,425.074,176.840,19.784,152.859
C08836=1092.276,232.849,425.100,176.837,19.782,152.859
C08837=1092.270,232.601,425.127,176.834,19.780,152.859
C08838=1092.264,232.352,425.152,176.831,19.778,152.859
C08839=1092.256,231.973,425.191,176.826,19.775,152.860
C08840=1092.248,231.594,425.231,176.822,19.772,152.860
C08841=1092.239,231.216,425.270,176.817,19.769,152.860
C08842=1092.231,230.837,425.309,176.813,19.766,152.860
C08843=1092.225,230.588,425.335,176.810,19.763,152.860
C08844=1092.219,230.339,425.360,176.807,19.762,152.860
C08845=1092.213,230.090,425.386,176.804,19.760,152.860
C08846=1092.208,229.841,425.412,176.801,19.758,152.860
C08847=1092.202,229.593,425.437,176.798,19.756,152.860
C08848=1092.197,229.344,425.463,176.795,19.755,152.861
C08849=1092.191,229.096,425.488,176.792,19.753,152.861
C08850=1092.185,228.847,425.514,176.789,19.750,152.861
C08851=1092.180,228.599,425.539,176.786,19.748,152.861
C08852=1092.174,228.350,425.565,176.783,19.746,152.861
C08853=1092.168,228.101,425.591,176.780,19.745,152.861
C08854=1092.163,227.853,425.616,176.777,19.743,152.861
C08855=1092.157,227.604,425.641,176.775,19.741,152.861
C08856=1092.151,227.355,425.667,176.771,19.739,152.861
C08857=1092.145,227.107,425.693,176.769,19.737,152.861
C08858=1092.140,226.858,425.718,176.766,19.735,152.861
C08859=1092.134,226.610,425.744,176.762,19.733,152.861
C08860=1092.129,226.361,425.770,176.760,19.731,152.862
C08861=1092.123,226.113,425.795,176.756,19.729,152.862
C08862=1092.118,225.863,425.820,176.754,19.727,152.862
C08863=1092.112,225.614,425.845,176.751,19.725,152.862
C08864=1092.107,225.366,425.871,176.748,19.723,152.862
C08865=1092.101,225.117,425.896,176.745,19.721,152.862
C08866=1092.095,224.868,425.922,176.742,19.720,152.862
C08867=1092.090,224.621,425.947,176.739,19.717,152.862
C08868=1092.084,224.371,425.972,176.737,19.716,152.862
C08869=1092.079,224.123,425.997,176.733,19.714,152.862
C08870=1092.073,223.874,426.022,176.731,19.712,152.862
C08871=1092.067,223.625,426.048,176.727,19.710,152.863
C08872=1092.062,223.377,426.073,176.724,19.707,152.863
C08873=1092.056,223.128,426.099,176.722,19.706,152.863
C08874=1092.051,222.880,426.124,176.718,19.704,152.863
C08875=1092.045,222.628,426.149,176.716,19.702,152.863
C08876=1092.039,222.376,426.175,176.712,19.700,152.863
C08877=1092.034,222.124,426.200,176.710,19.698,152.863
C08878=1092.028,221.873,426.226,176.707,19.696,152.863
C08879=1092.022,221.623,426.250,176.704,19.694,152.863
C08880=1092.017,221.375,426.276,176.701,19.692,152.863
C08881=1092.011,221.126,426.301,176.698,19.691,152.863
C08882=1092.005,220.877,426.326,176.695,19.689,152.863
C08883=1092.000,220.629,426.351,176.692,19.687,152.864
C08884=1091.994,220.379,426.376,176.689,19.685,152.864
C08885=1091.989,220.131,426.401,176.687,19.683,152.864
C08886=1091.983,219.883,426.426,176.683,19.681,152.864
C08887=1091.977,219.634,426.451,176.681,19.679,152.864
C08888=1091.972,219.385,426.477,176.677,19.677,152.864
C08889=1091.967,219.137,426.501,176.675,19.676,152.864
C08890=1091.960,218.888,426.526,176.672,19.674,152.864
C08891=1091.954,218.639,426.551,176.669,19.672,152.864
C08892=1091.949,218.391,426.576,176.666,19.669,152.864
C08893=1091.943,218.141,426.600,176.663,19.668,152.864
C08894=1091.938,217.893,426.626,176.660,19.666,152.865
C08895=1091.932,217.644,426.651,176.657,19.664,152.865
C08896=1091.927,217.396,426.675,176.654,19.662,152.865
C08897=1091.921,217.147,426.700,176.652,19.661,152.865
C08898=1091.915,216.898,426.724,176.648,19.658,152.865
C08899=1091.909,216.649,426.750,176.646,19.656,152.865
C08900=1091.905,216.400,426.775,176.643,19.654,152.865
C08901=1091.898,216.152,426.800,176.640,19.653,152.865
C08902=1091.893,215.903,426.824,176.637,19.651,152.865
C08903=1091.888,215.655,426.848,176.634,19.649,152.865
C08904=1091.882,215.406,426.874,176.631,19.647,152.866
C08905=1091.876,215.157,426.898,176.629,19.645,152.865
C08906=1091.870,214.908,426.923,176.625,19.643,152.866
C08907=1091.865,214.660,426.948,176.623,19.641,152.866
C08908=1091.860,214.410,426.973,176.619,19.639,152.866
C08909=1091.854,214.162,426.997,176.617,19.638,152.866
C08910=1091.849,213.914,427.022,176.613,19.636,152.866
C08911=1091.843,213.665,427.047,176.611,19.634,152.866
C08912=1091.837,213.416,427.071,176.608,19.631,152.866
C08913=1091.832,213.167,427.096,176.605,19.630,152.866
C08914=1091.826,212.918,427.120,176.602,19.628,152.866
C08915=1091.821,212.670,427.145,176.599,19.626,152.866
C08916=1091.815,212.421,427.169,176.597,19.625,152.867
C08917=1091.809,212.172,427.194,176.593,19.623,152.867
C08918=1091.804,211.923,427.218,176.591,19.621,152.867
C08919=1091.798,211.674,427.243,176.588,19.618,152.867
C08920=1091.793,211.426,427.267,176.585,19.617,152.867
C08921=1091.787,211.177,427.292,176.582,19.615,152.867
C08922=1091.781,210.929,427.316,176.579,19.613,152.867
C08923=1091.776,210.680,427.341,176.576,19.611,152.867
C08924=1091.770,210.431,427.365,176.573,19.610,152.867
C08925=1091.764,210.182,427.389,176.570,19.608,152.867
C08926=1091.758,209.933,427.414,176.568,19.605,152.867
C08927=1091.751,209.555,427.451,176.564,19.603,152.868
C08928=1091.742,209.177,427.488,176.559,19.600,152.868
C08929=1091.734,208.799,427.524,176.554,19.597,152.868
C08930=1091.725,208.420,427.562,176.550,19.595,152.868
C08931=1091.701,207.401,427.660,176.487,19.564,152.873
C08932=1091.696,207.152,427.684,176.484,19.564,152.873
C08933=1091.691,206.903,427.708,176.481,19.563,152.873
C08934=1091.684,206.654,427.732,176.478,19.562,152.874
C08935=1091.679,206.405,427.755,176.476,19.561,152.874
C08936=1091.674,206.156,427.780,176.472,19.559,152.874
C08937=1091.668,205.908,427.803,176.469,19.559,152.875
C08938=1091.663,205.659,427.828,176.466,19.558,152.875
C08939=1091.657,205.411,427.851,176.463,19.557,152.875
C08940=1091.651,205.161,427.875,176.460,19.556,152.875
C08941=1091.646,204.912,427.899,176.457,19.555,152.876
C08942=1091.640,204.664,427.922,176.454,19.554,152.876
C08943=1091.635,204.415,427.947,176.451,19.553,152.876
C08944=1091.629,204.166,427.970,176.448,19.552,152.877
C08945=1091.624,203.918,427.994,176.445,19.551,152.877
C08946=1091.618,203.669,428.018,176.442,19.550,152.877
C08947=1091.612,203.419,428.041,176.439,19.549,152.878
C08948=1091.607,203.171,428.066,176.437,19.548,152.878
C08949=1091.601,202.922,428.089,176.433,19.547,152.878
C08950=1091.596,202.673,428.113,176.430,19.546,152.879
C08951=1091.590,202.425,428.136,176.427,19.545,152.879
C08952=1091.585,202.176,428.160,176.424,19.544,152.879
C08953=1091.579,201.927,428.183,176.421,19.544,152.880
C08954=1091.572,201.678,428.207,176.419,19.543,152.880
C08955=1091.567,201.429,428.231,176.416,19.542,152.880
C08956=1091.561,201.181,428.254,176.413,19.541,152.880
C08957=1091.556,200.931,428.278,176.409,19.540,152.881
C08958=1091.550,200.683,428.301,176.406,19.539,152.881
C08959=1091.545,200.434,428.324,176.403,19.538,152.882
C08960=1091.539,200.186,428.349,176.400,19.537,152.882
C08961=1091.533,199.936,428.372,176.398,19.536,152.882
C08962=1091.527,199.687,428.395,176.395,19.535,152.882
C08963=1091.522,199.439,428.419,176.392,19.534,152.883
C08964=1091.516,199.190,428.442,176.389,19.534,152.883
C08965=1091.510,198.941,428.465,176.386,19.533,152.883
C08966=1091.505,198.692,428.489,176.382,19.531,152.884
C08967=1091.499,198.443,428.512,176.379,19.530,152.884
C08968=1091.493,198.195,428.536,176.377,19.529,152.884
C08969=1091.488,197.946,428.559,176.374,19.529,152.885
C08970=1091.483,197.697,428.582,176.371,19.528,152.885
C08971=1091.477,197.448,428.605,176.368,19.527,152.885
C08972=1091.472,197.199,428.630,176.365,19.526,152.886
C08973=1091.466,196.950,428.653,176.362,19.525,152.886
C08974=1091.460,196.702,428.676,176.359,19.524,152.886
C08975=1091.453,196.453,428.700,176.357,19.523,152.886
C08976=1091.449,196.203,428.723,176.354,19.523,152.887
C08977=1091.443,195.954,428.746,176.350,19.521,152.887
C08978=1091.437,195.706,428.769,176.347,19.520,152.887
C08979=1091.431,195.457,428.792,176.344,19.519,152.888
C08980=1091.426,195.208,428.816,176.342,19.518,152.888
C08981=1091.420,194.959,428.839,176.339,19.517,152.888
C08982=1091.415,194.710,428.862,176.336,19.516,152.889
C08983=1091.409,194.461,428.885,176.333,19.515,152.889
C08984=1091.404,194.213,428.908,176.330,19.514,152.889
C08985=1091.399,193.964,428.931,176.327,19.514,152.890
C08986=1091.393,193.716,428.955,176.324,19.513,152.890
C08987=1091.387,193.467,428.978,176.322,19.512,152.890
C08988=1091.382,193.218,429.001,176.319,19.511,152.890
C08989=1091.376,192.969,429.024,176.316,19.510,152.891
C08990=1091.370,192.720,429.047,176.312,19.508,152.891
C08991=1091.365,192.471,429.070,176.310,19.507,152.891
C08992=1091.358,192.195,429.096,176.307,19.507,152.892
C08993=1091.352,191.918,429.122,176.304,19.506,152.892
C08994=1091.346,191.642,429.147,176.300,19.504,152.892
C08995=1091.340,191.365,429.173,176.297,19.503,152.893
C08996=1091.335,191.116,429.195,176.294,19.502,152.893
C08997=1091.329,190.868,429.218,176.291,19.502,152.893
C08998=1091.324,190.618,429.242,176.289,19.501,152.893
C08999=1091.318,190.369,429.265,176.286,19.500,152.894
C09000=1091.313,190.121,429.288,176.282,19.498,152.894
C09001=1091.307,189.872,429.310,176.279,19.497,152.894
C09002=1091.302,189.624,429.333,176.276,19.496,152.895
C09003=1091.296,189.375,429.356,176.274,19.495,152.895
C09004=1091.291,189.125,429.380,176.271,19.494,152.895
C09005=1091.285,188.876,429.403,176.268,19.493,152.895
C09006=1091.279,188.628,429.426,176.265,19.492,152.896
C09007=1091.274,188.379,429.448,176.262,19.491,152.896
C09008=1091.269,188.131,429.471,176.260,19.490,152.896
C09009=1091.263,187.882,429.494,176.257,19.489,152.897
C09010=1091.257,187.632,429.516,176.254,19.488,152.897
C09011=1091.252,187.383,429.539,176.251,19.487,152.897
C09012=1091.247,187.134,429.563,176.248,19.486,152.898
C09013=1091.242,186.886,429.586,176.246,19.485,152.898
C09014=1091.236,186.637,429.608,176.243,19.484,152.898
C09015=1091.230,186.388,429.631,176.240,19.483,152.898
C09016=1091.225,186.138,429.654,176.237,19.482,152.899
C09017=1091.220,185.890,429.676,176.235,19.481,152.899
C09018=1091.214,185.641,429.699,176.232,19.480,152.899
C09019=1091.208,185.393,429.722,176.229,19.479,152.899
C09020=1091.203,185.143,429.744,176.226,19.478,152.900
C09021=1091.197,184.894,429.767,176.223,19.477,152.900
C09022=1091.191,184.645,429.790,176.220,19.476,152.900
C09023=1091.186,184.397,429.813,176.217,19.476,152.901
C09024=1091.180,184.148,429.834,176.215,19.475,152.901
C09025=1091.174,183.899,429.857,176.212,19.473,152.901
C09026=1091.168,183.650,429.880,176.209,19.473,152.901
C09027=1091.163,183.400,429.903,176.206,19.472,152.902
C09028=1091.157,183.152,429.926,176.203,19.471,152.902
C09029=1091.151,182.903,429.948,176.200,19.470,152.902
C09030=1091.146,182.654,429.970,176.198,19.469,152.903
C09031=1091.140,182.405,429.993,176.195,19.468,152.903
C09032=1091.134,182.157,430.015,176.192,19.467,152.903
C09033=1091.128,181.907,430.037,176.189,19.466,152.904
C09034=1091.123,181.658,430.060,176.186,19.465,152.904
C09035=1091.117,181.409,430.082,176.184,19.464,152.904
C09036=1091.111,181.161,430.104,176.181,19.463,152.904
C09037=1091.106,180.912,430.127,176.178,19.463,152.905
C09038=1091.100,180.662,430.150,176.175,19.461,152.905
C09039=1091.094,180.414,430.172,176.172,19.460,152.905
C09040=1091.089,180.165,430.194,176.169,19.459,152.906
C09041=1091.083,179.916,430.217,176.166,19.459,152.906
C09042=1091.078,179.667,430.239,176.164,19.458,152.906
C09043=1091.071,179.418,430.261,176.161,19.457,152.906
C09044=1091.066,179.169,430.284,176.158,19.456,152.907
C09045=1091.061,178.920,430.306,176.155,19.454,152.907
C09046=1091.055,178.671,430.328,176.152,19.454,152.907
C09047=1091.049,178.422,430.351,176.150,19.453,152.908
C09048=1091.044,178.173,430.373,176.147,19.452,152.908
C09049=1091.038,177.925,430.395,176.144,19.451,152.908
C09050=1091.032,177.675,430.417,176.141,19.450,152.908
C09051=1091.026,177.426,430.440,176.139,19.449,152.909
C09052=1091.021,177.178,430.461,176.136,19.448,152.909
C09053=1091.015,176.928,430.484,176.133,19.447,152.909
C09054=1091.009,176.680,430.506,176.130,19.446,152.910
C09055=1091.004,176.431,430.528,176.127,19.445,152.910
C09056=1090.997,176.154,430.552,176.124,19.444,152.910
C09057=1090.991,175.877,430.578,176.122,19.443,152.910
C09058=1090.985,175.601,430.602,176.118,19.441,152.911
C09059=1090.979,175.324,430.627,176.115,19.440,152.911
C09060=1090.973,175.075,430.649,176.112,19.439,152.911
C09061=1090.968,174.826,430.670,176.110,19.438,152.912
C09062=1090.962,174.578,430.693,176.107,19.437,152.912
C09063=1090.956,174.328,430.715,176.104,19.436,152.912
C09064=1090.952,174.079,430.737,176.101,19.435,152.912
C09065=1090.945,173.831,430.759,176.098,19.434,152.913
C09066=1090.940,173.581,430.781,176.096,19.433,152.913
C09067=1090.934,173.333,430.803,176.093,19.432,152.913
C09068=1090.929,173.083,430.825,176.090,19.431,152.913
C09069=1090.923,172.835,430.846,176.087,19.430,152.914
C09070=1090.917,172.586,430.869,176.084,19.429,152.914
C09071=1090.912,172.336,430.891,176.082,19.429,152.914
C09072=1090.906,172.088,430.913,176.080,19.428,152.914
C09073=1090.901,171.838,430.935,176.077,19.426,152.915
C09074=1090.895,171.590,430.956,176.074,19.425,152.915
C09075=1090.890,171.341,430.979,176.071,19.424,152.915
C09076=1090.884,171.092,431.001,176.069,19.423,152.915
C09077=1090.879,170.843,431.023,176.066,19.422,152.916
C09078=1090.873,170.594,431.044,176.063,19.421,152.916
C09079=1090.868,170.345,431.066,176.061,19.420,152.916
C09080=1090.862,170.096,431.088,176.058,19.418,152.916
C09081=1090.857,169.847,431.110,176.055,19.417,152.917
C09082=1090.851,169.598,431.131,176.052,19.416,152.917
C09083=1090.846,169.349,431.153,176.050,19.415,152.917
C09084=1090.840,169.100,431.175,176.047,19.414,152.917
C09085=1090.834,168.851,431.197,176.044,19.413,152.918
C09086=1090.828,168.602,431.219,176.042,19.413,152.918
C09087=1090.823,168.353,431.241,176.039,19.412,152.918
C09088=1090.817,168.104,431.262,176.037,19.410,152.918
C09089=1090.812,167.855,431.284,176.034,19.409,152.919
C09090=1090.806,167.606,431.306,176.031,19.408,152.919
C09091=1090.801,167.357,431.328,176.028,19.407,152.919
C09092=1090.795,167.108,431.349,176.026,19.406,152.919
C09093=1090.790,166.859,431.371,176.023,19.405,152.920
C09094=1090.785,166.609,431.392,176.020,19.404,152.920
C09095=1090.780,166.361,431.414,176.017,19.403,152.920
C09096=1090.774,166.111,431.436,176.015,19.401,152.920
C09097=1090.769,165.863,431.458,176.012,19.400,152.921
C09098=1090.763,165.614,431.479,176.010,19.399,152.921
C09099=1090.757,165.365,431.500,176.007,19.398,152.921
C09100=1090.752,165.116,431.522,176.005,19.397,152.921
C09101=1090.746,164.867,431.544,176.002,19.396,152.921
C09102=1090.741,164.618,431.566,175.999,19.395,152.922
C09103=1090.735,164.369,431.587,175.996,19.394,152.922
C09104=1090.731,164.119,431.609,175.994,19.392,152.922
C09105=1090.725,163.871,431.630,175.991,19.391,152.922
C09106=1090.719,163.622,431.652,175.988,19.390,152.923
